//Reset complete Fifo
METHOD PROTECTED _reset : BOOL //TRUE if method is finnished
VAR_INPUT
	pMemory													: 	POINTER TO BYTE := 0;
	SizeOfMemory											: 	UDINT := 0;
END_VAR
IF pMemory = 0
	OR SizeOfMemory = 0
THEN
	_reset													:= FALSE;
	RETURN;
ELSIF TestAndSet(Interlock)
THEN
	(* delete *)
	MEMSET(pMemory,0,SizeOfMemory);
	Empty 													:= TRUE;
	Full 													:= FALSE;
	Count 													:= 0;
	_reset													:= TRUE;
	Interlock												:= FALSE;
ELSE
	_reset													:= TRUE;
END_IF
END_METHOD

END_FUNCTION_BLOCK

// POUs/DataBuffer/Fifo/FifoExt
//FifoBase extended with dynamical memory allocation
 {attribute 'enable_dynamic_creation'}
FUNCTION_BLOCK FifoExt EXTENDS FifoBase
VAR_OUTPUT CONSTANT
END_VAR   
VAR_INPUT
	MaxNoOfEntrys											: 	UDINT := 10;	//0 = dynamically allocation / <> 0 = pre allcoation of memory based on size of first entry (n * data size) 
END_VAR
VAR_OUTPUT
	pMemory													: 	POINTER TO BYTE := 0; //Pointer to memory	
	SizeOfMemory											: 	UDINT := 0; //According MaxNoOfEntrys and SizeOfData of first entry
END_VAR
VAR
	MemSizeAllocatedMemory									:	UDINT := 0; //Allocated memory 
	MemSizeOfData											:	UDINT;
	MemMaxNoOfEntrys										:	UDINT;
	ExtInterlock											:	BOOL;
END_VAR

;

METHOD PROTECTED FINAL allocate : BOOL
VAR_IN_OUT
	SizeOfData												:	UDINT;
END_VAR
VAR
	pDummy													:	POINTER TO BYTE;	
End_Var
IF pMemory = 0
THEN
	IF SizeOfData = 0 OR MaxNoOfEntrys = 0
	THEN
		Allocate											:= FALSE;	
	ELSE
		MemSizeOfData										:= SizeOfData;
		MemMaxNoOfEntrys									:= MaxNoOfEntrys;
		SizeOfMemory										:= MemSizeOfData * MemMaxNoOfEntrys;
		MemSizeAllocatedMemory								:= SizeOfMemory;
		pMemory												:= __NEW(BYTE,SizeOfMemory );
		
		IF PARAM.ENABLE_DEBUG_MSG_DYNAMIC_MEM_ALLOCATION
		THEN
			AdsLogHint('EngineeringToolbox | FB FifoExt | An instance allocated %s bytes from the dynamic memory of the ADS router memory pool', TO_STRING(SizeOfMemory));
		END_IF
	END_IF

ELSIF SizeOfData = MemSizeOfData AND MaxNoOfEntrys = MemMaxNoOfEntrys
THEN
	Allocate												:= TRUE;
	
ELSIF SizeOfData > MemSizeOfData OR MaxNoOfEntrys > MemMaxNoOfEntrys
THEN //Since increased, allocate new memory
	MemSizeAllocatedMemory									:= SizeOfData * MaxNoOfEntrys;
	pDummy													:= __NEW(BYTE, MemSizeAllocatedMemory); 
	
	 //Size of data still the same, copy old data to reuse
	IF MemSizeOfData = SizeOfData AND Count > 0
	THEN
		MEMCPY(pDummy,pMemory, SizeOfMemory);
	END_IF
	
	//Copy new settings to local variales
	MemSizeOfData											:= SizeOfData;
	MemMaxNoOfEntrys										:= MaxNoOfEntrys;	
	SizeOfMemory 											:= MemSizeAllocatedMemory;

	__DELETE(pMemory);  //Delete reference to old memory
	pMemory													:= pDummy; //Take over new pointer to new memory
	
	IF PARAM.ENABLE_DEBUG_MSG_DYNAMIC_MEM_ALLOCATION
	THEN
		AdsLogWarn('EngineeringToolbox | FB FifoExt | Value of "MaxNoOfEntrys" or data size increased and one instance allocated additional %s bytes from the dynamic memory of the ADS router memory pool', TO_STRING(SizeOfMemory));
	END_IF
	
	Allocate												:= TRUE;
	
ELSE //Size decreased
	IF MemSizeOfData <> SizeOfData AND Count > 0
	THEN //Size of data changed, erease memory 
		MEMSET(pMemory,0, MemSizeAllocatedMemory);
	ELSE //Size of data the same, keep current data
		;
	END_IF
	
	//Copy new settings to local variales
	MemSizeOfData											:= SizeOfData;
	MemMaxNoOfEntrys										:= MaxNoOfEntrys;
	SizeOfMemory											:= MemSizeOfData * MemMaxNoOfEntrys;
	Allocate												:= TRUE;
END_IF
END_METHOD

//Clear out one entry from the Fifo buffer
METHOD PUBLIC clear : BOOL //TRUE if method was successful
VAR_INPUT
	EntryNo													:	UDINT;
END_VAR             										
VAR                 										
END_VAR
Clear := SUPER^._Clear(EntryNo,This^.pMemory,This^.SizeOfMemory);
END_METHOD

//Clear out defined data set from the Fifo buffer
METHOD PUBLIC clearByDataSet : BOOL //TRUE if method was successful
VAR_INPUT
	pData													: 	POINTER TO BYTE := 0;				
END_VAR             										
VAR                 										
END_VAR
ClearByDataSet := SUPER^._ClearByDataSet(pData,SizeOfEntry,This^.pMemory,This^.SizeOfMemory);
END_METHOD

METHOD PUBLIC dequeue : BOOL //TRUE if method was successful
VAR_INPUT
	pData													:	POINTER TO BYTE;	
END_VAR
VAR
END_VAR
Dequeue := SUPER^._Dequeue(pData,SizeOfEntry,This^.pMemory,This^.SizeOfMemory);
END_METHOD

METHOD PUBLIC enqueue : BOOL //TRUE if method was successful
VAR_INPUT
	pData													:	POINTER TO BYTE;
	SizeOfData												:	UDINT;
END_VAR
VAR
	CopySize												:	UDINT;
	pDummy													:	POINTER TO BYTE;
END_VAR
IF TestAndSet(ExtInterlock) 
THEN	
	if Allocate(SizeOfData)
	then
		Enqueue 											:= SUPER^._Enqueue(pData,SizeOfData,THIS^.pMemory,THIS^.SizeOfMemory);
		ExtInterlock										:= FALSE;
	else
		Enqueue												:= FALSE;
	END_IF	
ELSE
	Enqueue													:= FALSE;
END_IF
END_METHOD

METHOD FB_exit : BOOL
VAR_INPUT
	bInCopyCode : BOOL; // if TRUE, the exit method is called for exiting an instance that is copied afterwards (online change).
END_VAR
IF NOT bInCopyCode AND pMemory <> 0
THEN //Release memory in case the PLC stopps
	__DELETE(pMemory);
	Full													:= FALSE;
	Empty													:= TRUE;
	Count													:= 0;
	SizeOfMemory											:= 0;
	MemSizeOfData											:= 0;
	MemSizeAllocatedMemory									:= 0;
	MemMaxNoOfEntrys										:= MaxNoOfEntrys;
END_IF
END_METHOD

//Check wheter a value already exist
METHOD PUBLIC isEnqueued : UDINT //pData entry exist in Fifo at idx as return value 
VAR_INPUT
	pData													: 	POINTER TO BYTE := 0;
END_VAR
IsEnqueued := SUPER^._IsEnqueued(pData,SizeOfEntry,This^.pMemory,This^.SizeOfMemory);
END_METHOD

//Check wheter a value will be the next output of the buffer
METHOD PUBLIC isNextEntry : BOOL //Inputs value is the next output 
VAR_INPUT
	pData													: 	POINTER TO BYTE := 0;
END_VAR
VAR
END_VAR
IsNextEntry := SUPER^._IsNextEntry(pData,SizeOfEntry,This^.pMemory,This^.SizeOfMemory);
END_METHOD

METHOD PUBLIC readEntry : BOOL //TRUE if method was successful
VAR_INPUT
	idx														:	UDINT;
	pData													: 	POINTER TO BYTE := 0;
END_VAR
ReadEntry := SUPER^._ReadEntry(idx,pData,SizeOfEntry,This^.pMemory,This^.SizeOfMemory);
END_METHOD

//Reset complete Fifo
METHOD PUBLIC reset : BOOL //TRUE if method is finnished
VAR_INPUT
END_VAR
reset				:= SUPER^._reset(This^.pMemory,This^.SizeOfMemory);
END_METHOD

END_FUNCTION_BLOCK

// POUs/DataBuffer/Fifo/FifoLRealSimple
//Fifo with a internal Lreal array for a simple num list implementation
FUNCTION_BLOCK FifoLRealSimple EXTENDS FifoBase
VAR_OUTPUT CONSTANT
	MIN_BUFFER												:	DINT := 1; //Fifo buffer start index 
	MAX_BUFFER												:	DINT := PARAM.FIFO_LREAL_SIMPEL_MAX_BUFFER; //Fifo buffer end index - see library parameter to customize parameter
END_VAR   
VAR_INPUT
END_VAR
VAR_OUTPUT
	Buffer													:	ARRAY[MIN_BUFFER..MAX_BUFFER] OF LREAL; //Lreal Fifo buffer 
END_VAR
VAR
END_VAR

;

 //Clear out one entry from the Fifo buffer
METHOD PUBLIC clear : BOOL //TRUE if method was successful
VAR_INPUT
	EntryNo													:	UDINT;
END_VAR             										
VAR                 										
END_VAR
Clear := super^._Clear(EntryNo,ADR(Buffer),SIZEOF(Buffer));
END_METHOD

//Clear out defined data set from the Fifo buffer
METHOD PUBLIC clearByDataSet : BOOL //TRUE if method was successful
VAR_INPUT
	Value													:	LREAL;
END_VAR             										
VAR                 										
END_VAR
ClearByDataSet := super^._ClearByDataSet(ADR(Value),SIZEOF(Value),ADR(Buffer),SIZEOF(Buffer));
END_METHOD

METHOD PUBLIC dequeue : BOOL //TRUE if method was successful
VAR_IN_OUT
	Value													:	LREAL;	
END_VAR
VAR
END_VAR
Dequeue := SUPER^._Dequeue(ADR(Value),SIZEOF(Value),ADR(Buffer),SIZEOF(Buffer));
END_METHOD

METHOD PUBLIC enqueue : BOOL //TRUE if method was successful
VAR_INPUT
	Value													:	LREAL;
END_VAR
Enqueue := SUPER^._Enqueue(ADR(Value),SIZEOF(Value),ADR(Buffer),SIZEOF(Buffer));
END_METHOD

//Check wheter a value already exist
METHOD PUBLIC isEnqueued : uDINT //In Value exist in Fifo at idx as return value  
VAR_INPUT
	Value													:	LREAL;
END_VAR
IsEnqueued := SUPER^._IsEnqueued(ADR(Value),SIZEOF(Value),ADR(Buffer),SIZEOF(Buffer));
END_METHOD

//Check wheter a value will be the next output of the buffer
METHOD PUBLIC isNextEntry : BOOL //Inputs value is the next output 
VAR_INPUT
	Value													: LREAL;
END_VAR
VAR
END_VAR
IsNextEntry := SUPER^._IsNextEntry(ADR(Value),SIZEOF(Value),ADR(Buffer),SIZEOF(Buffer));
END_METHOD

METHOD PUBLIC readEntry : BOOL //TRUE if method was successful
VAR_INPUT
	idx														:	uDINT;
END_VAR
VAR_IN_OUT
	value													: LREAL;	
END_VAR
ReadEntry := SUPER^._ReadEntry(idx,ADR(Value),SIZEOF(Value),ADR(Buffer),SIZEOF(Buffer));
END_METHOD

//Reset complete Fifo
METHOD PUBLIC reset : BOOL //TRUE if method is finnished
VAR_INPUT
END_VAR
reset := SUPER^._reset(ADR(Buffer),SIZEOF(Buffer));
END_METHOD

END_FUNCTION_BLOCK

// POUs/DataBuffer/Ringbuffer/Ringbuffer
//Ringbuffer based on external memory
FUNCTION_BLOCK Ringbuffer EXTENDS RingbufferBase
VAR_INPUT	
END_VAR
VAR_OUTPUT
END_VAR    
VAR
END_VAR

METHOD PUBLIC dequeue : BOOL //TRUE if method was successful
VAR_INPUT
	pData													: 	POINTER TO BYTE ;
	SizeOfData												: 	UDINT ;
	pMemory													: 	POINTER TO BYTE ;
	SizeOfMemory											: 	UDINT ;
END_VAR
Dequeue := SUPER^._Dequeue(pData,SizeOfData,pMemory,SizeOfMemory);
END_METHOD

METHOD PUBLIC dequeueStream : BOOL //TRUE if method was successful
VAR_INPUT
	pData													: 	POINTER TO BYTE ;
	SizeOfStream											:	UDINT ; //n * Size of last entry and not greater than SizeOfMemory
	pMemory													: 	POINTER TO BYTE;
	SizeOfMemory											: 	UDINT ;
END_VAR
VAR
END_VAR
DequeueStream := SUPER^._DequeueStream(pData,SizeOfStream,pMemory,SizeOfMemory);
END_METHOD

METHOD PUBLIC enqueue : BOOL //TRUE if method was successful
VAR_INPUT
	pData													: 	POINTER TO BYTE ;
	SizeOfData												: 	UDINT ;
	pMemory													: 	POINTER TO BYTE ;
	SizeOfMemory											: 	UDINT ;
END_VAR
Enqueue := SUPER^._Enqueue(pData,SizeOfData,pMemory,SizeOfMemory);
END_METHOD

METHOD PUBLIC enqueueStream : BOOL
VAR_INPUT
	pData													: 	POINTER TO BYTE ;
	SizeOfData												: 	UDINT ; //Size of one entry
	SizeOfStream											:	UDINT ; //n * SizeofData and not greater than SizeOfMemory
	pMemory													: 	POINTER TO BYTE ;
	SizeOfMemory											: 	UDINT ;
END_VAR
VAR
END_VAR
EnqueueStream := SUPER^._EnqueueStream(pData,SizeOfData,SizeOfStream,pMemory,SizeOfMemory);
END_METHOD

//Reset complete ring buffer
METHOD PUBLIC reset : BOOL //TRUE if method is finnished
VAR_INPUT
	pMemory													: 	POINTER TO BYTE := 0;
	SizeOfMemory											: 	UDINT := 0;
END_VAR
reset := SUPER^._reset(pMemory,SizeOfMemory);
END_METHOD

END_FUNCTION_BLOCK

// POUs/DataBuffer/Ringbuffer/RingbufferBase
//Ringbuffer basic template based on external memory
FUNCTION_BLOCK RingbufferBase
VAR_INPUT	
	Overwrite												:	BOOL := FALSE; // TRUE = overwrite oldest entry 
END_VAR
VAR_OUTPUT
	Count													:	UDINT := 0; 	// Number of entrys	
	Full													:	BOOL ;		// TRUE when max number of entrys reached
	Empty													:	BOOL := TRUE; // TRUE when no entrys present
	ReadIdx													: 	UDINT := 0;	// Read data from adress 
	WriteIdx												: 	UDINT := 0;	// Write data to adress
END_VAR    
VAR
	Interlock												:	BOOL; 
	MaxEntrys												:	UDINT; //Maximum number of entrys based on size of data and size of memory
	SizeOfEntry												:	UDINT;
	NoOfStreamEntrys										:	UDINT;
	cbData													:	UDINT;
END_VAR

METHOD PROTECTED _dequeue : BOOL //TRUE if method was successful
VAR_INPUT
	pData													: 	POINTER TO BYTE ;
	SizeOfData												: 	UDINT ;
	pMemory													: 	POINTER TO BYTE ;
	SizeOfMemory											: 	UDINT ;
END_VAR
IF 	pData = 0
	OR SizeOfData = 0
	OR pMemory = 0
	OR SizeOfMemory = 0
	OR Empty
THEN
	_Dequeue												:= FALSE;
	RETURN;
ELSIF TestAndSet(Interlock)
THEN	
	IF Count > 0
	THEN 
		(* copy dataset *)
		ReadIdx												:= ReadIdx + 1;
		IF (ReadIdx) > MaxEntrys
		THEN
			ReadIdx											:= 1;						
		END_IF
		
		MEMCPY(pData,pMemory + MAX(0, ReadIdx - 1) * SizeOfData,SizeOfData);
		
		Count 												:= MAX(0,Count - 1);
		Empty 												:= Count = 0;
		Full												:= FALSE;
		_Dequeue											:= TRUE;	
	ELSE 
		_Dequeue											:= FALSE;
	END_IF
	
	Interlock												:= FALSE;
ELSE
	_Dequeue												:= FALSE;
END_IF
END_METHOD

METHOD PROTECTED _dequeueStream : BOOL //TRUE if method was successful
VAR_INPUT
	pData													: 	POINTER TO BYTE ;
	SizeOfStream											:	UDINT ; //n * Size of last entry and not greater than SizeOfMemory
	pMemory													: 	POINTER TO BYTE;
	SizeOfMemory											: 	UDINT ;
END_VAR
VAR
END_VAR
IF 	pData = 0
	OR SizeOfEntry = 0
	OR pMemory = 0
	OR SizeOfMemory = 0
	OR Empty 
	OR SizeOfStream > SizeOfMemory
THEN
	_DequeueStream											:= FALSE;
	RETURN;
ELSIF TestAndSet(Interlock)
THEN	
	NoOfStreamEntrys										:= (SizeOfStream / SizeOfEntry); 
	IF Count > 0  
	THEN 
		(* maximum count *)
		IF ReadIdx + MIN(Count,NoOfStreamEntrys) <= MaxEntrys
		THEN //Read all data at one time
			ReadIdx											:= ReadIdx + 1; //Point to start read data			
			MEMCPY(pData,pMemory + (ReadIdx - 1) * SizeOfEntry, MIN(TO_UDINT(Count) * SizeOfEntry, SizeOfStream));
			ReadIdx											:= (ReadIdx - 1) + TO_UDINT(MIN(Count, NoOfStreamEntrys)); //Point to next index after reading x entrys
				
		ELSE //Read data with overflow					
			cbData											:= TO_UDINT(MaxEntrys) - ReadIdx; 		 
			ReadIdx											:= ReadIdx + 1; //Point to start read data	
			//Copy first part of stream our from buffer
			MEMCPY(pData, pMemory + ((ReadIdx - 1) * SizeOfEntry), cbData * SizeOfEntry );
	
			//Copy second part of stream from beginning of buffer
			ReadIdx											:= TO_UDINT(MIN(Count,NoOfStreamEntrys)) - cbData; //Point to next index after reading x entrys	
			MEMCPY( pData + (cbData * SizeOfEntry) , pMemory ,(TO_UDINT(MIN(Count,NoOfStreamEntrys)) - cbData) * SizeOfEntry);			
		END_IF
		Count 												:= MAX(0,Count - NoOfStreamEntrys);		
		Empty 												:= Count = 0;
		Full												:= FALSE;
		_DequeueStream										:= TRUE;	
		
	ELSE 
		_DequeueStream										:= FALSE;
	END_IF
	
	Interlock												:= FALSE;
ELSE
	_DequeueStream											:= FALSE;
END_IF
END_METHOD

METHOD PROTECTED _enqueue : BOOL //TRUE if method was successful
VAR_INPUT
	pData													: 	POINTER TO BYTE ;
	SizeOfData												: 	UDINT ;
	pMemory													: 	POINTER TO BYTE ;
	SizeOfMemory											: 	UDINT ;
END_VAR
IF pData = 0
	OR SizeOfData = 0
	OR pMemory = 0
	OR SizeOfMemory = 0
THEN
	_Enqueue												:= FALSE;
	RETURN;
ELSIF TestAndSet(Interlock)
THEN			
	_Enqueue												:= FALSE;
	
	(* maximum count *)
	MaxEntrys 												:= (SizeOfMemory / SizeOfData);

	IF Count < MaxEntrys OR Overwrite
	THEN
		SizeOfEntry											:= SizeOfData;
		IF MaxEntrys = Count 
		THEN //Adapt read index if write index is in front of read index
			ReadIdx											:= ReadIdx + 1;
			IF ReadIdx > TO_UDINT(MaxEntrys)
			THEN
				ReadIdx										:= 1;								
			END_IF
		END_IF	
		WriteIdx											:= WriteIdx + 1;	
		IF WriteIdx > TO_UDINT(MaxEntrys)
		THEN
			WriteIdx										:= 1;
		END_IF
	
		MEMCPY(pMemory + ((MAX(0,WriteIdx) - 1) * SizeOfData) ,pData,SizeOfData);		
		Count												:= MIN(Count + 1,  MaxEntrys);
		Full												:= Count >= MaxEntrys;
		Empty 												:= FALSE;	
		_Enqueue											:= TRUE;
	END_IF
	
	Interlock												:= FALSE;
ELSE
	_Enqueue												:= FALSE;
END_IF
END_METHOD

METHOD PROTECTED _enqueueStream : BOOL
VAR_INPUT
	pData													: 	POINTER TO BYTE ;
	SizeOfData												: 	UDINT ; //Size of one entry
	SizeOfStream											:	UDINT ; //n * SizeofData and not greater than SizeOfMemory
	pMemory													: 	POINTER TO BYTE ;
	SizeOfMemory											: 	UDINT ;
END_VAR
VAR
END_VAR
IF pData = 0
	OR SizeOfData = 0
	OR pMemory = 0
	OR SizeOfMemory = 0
	OR SizeOfStream = 0
	OR SizeOfStream > SizeOfMemory 
THEN
	_EnqueueStream											:= FALSE;
	RETURN;
ELSIF TestAndSet(Interlock)
THEN			
	_EnqueueStream											:= FALSE;
	
	(* maximum count *)
	MaxEntrys 												:= (SizeOfMemory / SizeOfData);
	SizeOfEntry												:= SizeOfData;
	NoOfStreamEntrys										:= (SizeOfStream / SizeOfData);
	
	IF (WriteIdx) + NoOfStreamEntrys <= MaxEntrys
	THEN //write full stream
		IF Count < MaxEntrys OR Overwrite
		THEN
			IF MaxEntrys = Count
			THEN //Adapt read index if write index is in front of read index
				ReadIdx										:= ReadIdx + TO_UDINT(NoOfStreamEntrys); 			
			END_IF		
		
			MEMCPY(pMemory + (WriteIdx * SizeOfData) ,pData,SizeOfStream);		
			WriteIdx										:= writeIdx + TO_UDINT(NoOfStreamEntrys);
			Count											:= MIN(Count + NoOfStreamEntrys, MaxEntrys);
			Empty 											:= FALSE;	
			_EnqueueStream									:= TRUE;
		ELSE
			_EnqueueStream									:= FALSE;
		END_IF	
	ELSIF Count + NoOfStreamEntrys <= (MaxEntrys) OR Overwrite
	THEN //Stream causes overflow
		cbData												:= TO_UDINT(MaxEntrys) - WriteIdx; 		 
		//Copy first part of stream to fill up buffer
		MEMCPY(pMemory + (WriteIdx * SizeOfData) ,pData, (cbData * SizeOfData) );	
		//Copy second part of stream to beginning of buffer
		MEMCPY(pMemory , pData + (cbData * SizeOfData) ,(TO_UDINT(NoOfStreamEntrys) - cbData) * SizeOfData);	
		
		WriteIdx											:= (writeIdx + TO_UDINT(NoOfStreamEntrys)) - TO_UDINT(MaxEntrys);
		Count												:= MIN(Count + NoOfStreamEntrys, MaxEntrys);
		IF MaxEntrys = Count
		THEN //Adapt read index if write index is in front of read index
			ReadIdx											:= WriteIdx;
		END_IF	
			
		Empty 												:= FALSE;	
		_EnqueueStream										:= TRUE;	
	ELSE
		_EnqueueStream										:= FALSE;	
	END_IF		
	Full													:= Count >= MaxEntrys;
	Interlock												:= FALSE;
ELSE
	_EnqueueStream											:= FALSE;
END_IF
END_METHOD

//Reset complete ring buffer
METHOD PROTECTED _reset : BOOL //TRUE if method is finnished
VAR_INPUT
	pMemory													: 	POINTER TO BYTE := 0;
	SizeOfMemory											: 	UDINT := 0;
END_VAR
IF pMemory = 0
	OR SizeOfMemory = 0
THEN
	_reset													:= TRUE;
	RETURN;
ELSIF TestAndSet(Interlock)
THEN
	(* delete *)
	_reset													:= TRUE;
	MEMSET(pMemory,0,SizeOfMemory);
	ReadIdx := WriteIdx										:= 0;
	Empty 													:= TRUE;
	Full													:= FALSE;
	Count 													:= 0;
	Interlock												:= FALSE;
ELSE
	_reset													:= TRUE;
END_IF
END_METHOD

END_FUNCTION_BLOCK

// POUs/DataBuffer/Ringbuffer/RingbufferByteSimple
//Ringbuffer with a internal Byte array for a simple data buffer implementation 
FUNCTION_BLOCK RingbufferByteSimple EXTENDS RingbufferBase
VAR_OUTPUT CONSTANT
	MIN_BUFFER												:	UDINT := 1; //Ringbuffer start index 
	MAX_BUFFER												:	uDINT := PARAM.RINGBUFFER_BYTE_SIMPLE_MAX_BUFFER; //Ringbuffer buffer end index - see library parameter to customize parameter
END_VAR   
VAR_INPUT
END_VAR
VAR_OUTPUT
	Buffer													:	ARRAY[MIN_BUFFER..MAX_BUFFER] OF BYTE; //Byte buffer 
END_VAR
VAR 
END_VAR

;

METHOD PUBLIC dequeue : BOOL //TRUE if method was successful
VAR_IN_OUT
	value													: BYTE;	
END_VAR
IF TestAndSet(Interlock)
THEN	
	IF Count > 0
	THEN 
		(* copy dataset *)		
		ReadIdx												:= ReadIdx + 1;
		IF (ReadIdx) > MAX_BUFFER
		THEN
			ReadIdx											:= TO_UDINT(MIN_BUFFER);				
		END_IF
		
		Value												:= Buffer[ReadIdx];
		
		Count 												:= MAX(0,Count - 1);
		Empty 												:= Count = 0;
		Full												:= FALSE;
		Dequeue												:= TRUE;	
	ELSE 
		Dequeue												:= FALSE;
	END_IF
	
	Interlock												:= FALSE;
ELSE
	Dequeue													:= FALSE;
END_IF
END_METHOD

METHOD PUBLIC dequeueStream : BOOL //TRUE if method was successful
VAR_INPUT
	pData													:	POINTER TO BYTE;
	SizeOfStream											:	UDINT;	
END_VAR
DequeueStream := super^._DequeueStream(pData, SizeOfStream,  ADR(Buffer),SIZEOF(Buffer));
END_METHOD

METHOD PUBLIC enqueue : BOOL //TRUE if method was successful
VAR_INPUT
	Value													:	BYTE;
END_VAR
IF TestAndSet(Interlock)
THEN			
	Enqueue													:= FALSE;

	IF Count < MAX_BUFFER OR Overwrite
	THEN
		IF MAX_BUFFER = Count 
		THEN //Adapt read index if write index is in front of read index
			ReadIdx											:= ReadIdx + 1;
			IF ReadIdx > TO_UDINT(MAX_BUFFER)
			THEN
				ReadIdx										:= TO_UDINT(MIN_BUFFER);							
			END_IF
		END_IF		
		WriteIdx											:= WriteIdx + 1;	
		IF WriteIdx > TO_UDINT(MAX_BUFFER)
		THEN
			WriteIdx										:= TO_UDINT(MIN_BUFFER);
		END_IF
	
		Buffer[WriteIdx]									:= Value;
	
		Count												:= MIN(Count + 1,  MAX_BUFFER);
		Full												:= Count >= MAX_BUFFER;
		Empty 												:= FALSE;	
		Enqueue												:= TRUE;
	END_IF
	
	Interlock												:= FALSE;
ELSE
	Enqueue													:= FALSE;
END_IF
END_METHOD

METHOD PUBLIC enqueueStream : BOOL //TRUE if method was successful
VAR_INPUT
	pData													:	POINTER TO BYTE;
	SizeOfStream											:	UDINT;
END_VAR
EnqueueStream := SUPER^._EnqueueStream(pData, SIZEOF(BUFFER[MIN_BUFFER] ), SizeOfStream,ADR(Buffer),SIZEOF(Buffer));
END_METHOD

//Reset complete ring buffer
METHOD PUBLIC reset : BOOL //TRUE if method is finnished
VAR_INPUT
END_VAR
reset := SUPER^._reset(ADR(Buffer),SIZEOF(Buffer));
END_METHOD

END_FUNCTION_BLOCK

// POUs/DataBuffer/Ringbuffer/RingbufferCharSimple
//Ringbuffer with a internal char array (String) for a simple num list implementation
FUNCTION_BLOCK RingbufferCharSimple EXTENDS RingbufferBase
VAR_OUTPUT CONSTANT
	MIN_BUFFER												:	UDINT := 0; //Default min index of string 
	MAX_BUFFER												:	UDINT := PARAM.RINGBUFFER_CHAR_SIMPLE_MAX_BUFFER; //Ringbuffer buffer end index - see library parameter to customize parameter
END_VAR   
VAR_INPUT
END_VAR
VAR_OUTPUT
	Buffer													:	STRING[MAX_BUFFER]; //Char buffer 
END_VAR
VAR
END_VAR

;

METHOD PUBLIC dequeue : BOOL //TRUE if method was successful
VAR_IN_OUT
	value													: BYTE;	
END_VAR
Dequeue := SUPER^._Dequeue(ADR(Value),SizeOfEntry,ADR(Buffer),SIZEOF(Buffer));
END_METHOD

METHOD PUBLIC dequeueStream : BOOL //TRUE if method was successful
VAR_INPUT
	pData													:	POINTER TO BYTE;
	SizeOfStream											:	UDINT ; //Not greater than SizeOfMemory
END_VAR
DequeueStream := SUPER^._DequeueStream(pData, SizeOfStream,  ADR(Buffer),TO_UDINT(MAX_BUFFER));
END_METHOD

METHOD PUBLIC enqueue : BOOL //TRUE if method was successful
VAR_INPUT
	Value													:	BYTE;
END_VAR
Enqueue := SUPER^._Enqueue(ADR(Value),SIZEOF(Value),ADR(Buffer),SIZEOF(Buffer));
END_METHOD

METHOD PUBLIC enqueueStream : BOOL //TRUE if method was successful
VAR_INPUT
	pData													:	POINTER TO BYTE;
	SizeOfStream											:	UDINT ; //Not greater than SizeOfMemory
END_VAR
EnqueueStream := SUPER^._EnqueueStream(pData,SIZEOF(BUFFER[MIN_BUFFER]), SizeOfStream,ADR(Buffer),TO_UDINT(MAX_BUFFER));
END_METHOD

//Reset complete ring buffer
METHOD PUBLIC reset : BOOL //TRUE if method is finnished
VAR_INPUT
END_VAR
reset := SUPER^._reset(ADR(Buffer),SIZEOF(Buffer));
END_METHOD

END_FUNCTION_BLOCK

// POUs/DataBuffer/Ringbuffer/RingbufferExt
//Ringbuffer extended with dynamical allocation of memory 
{attribute 'enable_dynamic_creation'}
FUNCTION_BLOCK RingbufferExt EXTENDS RingbufferBase
VAR_OUTPUT CONSTANT
END_VAR   
VAR_INPUT
	MaxNoOfEntrys											: 	UDINT := 10;	//0 = dynamically allocation / <> 0 = pre allcoation of memory based on size of first entry (n * data size) 
END_VAR
VAR_OUTPUT
	pMemory													: 	POINTER TO BYTE := 0;	//start address of buffer data
	SizeOfMemory											: 	UDINT := 0;	//size of buffer
END_VAR
VAR
	MemSizeAllocatedMemory									:	UDINT := 0; //Allocated memory 
	MemSizeOfData											:	UDINT;
	MemMaxNoOfEntrys										:	UDINT;
	ExtInterlock											:	BOOL;
END_VAR

;

METHOD PROTECTED FINAL allocate : BOOL
VAR_IN_OUT
	SizeOfData												:	UDINT;
END_VAR
VAR
	pDummy													:	POINTER TO BYTE;	
End_Var
IF pMemory = 0
THEN
	IF SizeOfData = 0 OR MaxNoOfEntrys = 0
	THEN
		Allocate											:= FALSE;	
	ELSE
		MemSizeOfData										:= SizeOfData;
		MemMaxNoOfEntrys									:= MaxNoOfEntrys;
		SizeOfMemory										:= MemSizeOfData * MemMaxNoOfEntrys;
		MemSizeAllocatedMemory								:= SizeOfMemory;
		pMemory												:= __NEW(BYTE,SizeOfMemory );
		
		IF PARAM.ENABLE_DEBUG_MSG_DYNAMIC_MEM_ALLOCATION
		THEN
			AdsLogHint('EngineeringToolbox | FB FifoExt | An instance allocated %s bytes from the dynamic memory of the ADS router memory pool', TO_STRING(SizeOfMemory));
		END_IF
	END_IF

ELSIF SizeOfData = MemSizeOfData AND MaxNoOfEntrys = MemMaxNoOfEntrys
THEN
	Allocate												:= TRUE;
	
ELSIF SizeOfData > MemSizeOfData OR MaxNoOfEntrys > MemMaxNoOfEntrys
THEN //Since increased, allocate new memory
	MemSizeAllocatedMemory									:= SizeOfData * MaxNoOfEntrys;
	pDummy													:= __NEW(BYTE, MemSizeAllocatedMemory); 
	
	 //Size of data still the same, copy old data to reuse
	IF MemSizeOfData = SizeOfData AND Count > 0
	THEN
		MEMCPY(pDummy,pMemory, SizeOfMemory);
	END_IF
	
	//Copy new settings to local variales
	MemSizeOfData											:= SizeOfData;
	MemMaxNoOfEntrys										:= MaxNoOfEntrys;	
	SizeOfMemory 											:= MemSizeAllocatedMemory;

	__DELETE(pMemory);  //Delete reference to old memory
	pMemory													:= pDummy; //Take over new pointer to new memory
	
	IF PARAM.ENABLE_DEBUG_MSG_DYNAMIC_MEM_ALLOCATION
	THEN
		AdsLogWarn('EngineeringToolbox | FB FifoExt | Value of "MaxNoOfEntrys" or data size increased and one instance allocated additional %s bytes from the dynamic memory of the ADS router memory pool', TO_STRING(SizeOfMemory));
	END_IF
	
	Allocate												:= TRUE;
	
ELSE //Size decreased
	IF MemSizeOfData <> SizeOfData AND Count > 0
	THEN //Size of data changed, erease memory 
		MEMSET(pMemory,0, MemSizeAllocatedMemory);
	ELSE //Size of data the same, keep current data
		;
	END_IF
	
	//Copy new settings to local variales
	MemSizeOfData											:= SizeOfData;
	MemMaxNoOfEntrys										:= MaxNoOfEntrys;
	SizeOfMemory											:= MemSizeOfData * MemMaxNoOfEntrys;
	Allocate												:= TRUE;
END_IF
END_METHOD

METHOD PUBLIC dequeue : BOOL //TRUE if method was successful
VAR_INPUT
	pData													:	POINTER TO BYTE;	
END_VAR
VAR
END_VAR
Dequeue := SUPER^._Dequeue(pData,SizeOfEntry,This^.pMemory,This^.SizeOfMemory);
END_METHOD

METHOD PUBLIC dequeueStream : BOOL //TRUE if method was successful
VAR_INPUT
	pData													:	POINTER TO BYTE;	
	SizeOfStream											:	UDINT ; //Not greater than SizeOfMemory
END_VAR
VAR
END_VAR
DequeueStream := SUPER^._DequeueStream(pData,SizeOfStream , This^.pMemory,This^.SizeOfMemory);
END_METHOD

METHOD PUBLIC enqueue : BOOL //TRUE if method was successful
VAR_INPUT
	pData													:	POINTER TO BYTE;
	SizeOfData												:	UDINT;
END_VAR
VAR
END_VAR
IF TestAndSet(ExtInterlock) 
THEN	
	if Allocate(SizeOfData)
	then
		Enqueue 											:= SUPER^._Enqueue(pData,SizeOfData,THIS^.pMemory,THIS^.SizeOfMemory);
		ExtInterlock										:= FALSE;
	else
		Enqueue												:= FALSE;
	END_IF	
ELSE
	Enqueue													:= FALSE;
END_IF
END_METHOD

METHOD PUBLIC enqueueStream : BOOL //TRUE if method was successful
VAR_INPUT
	pData													:	POINTER TO BYTE;
	SizeOfData												:	UDINT; //Size of one entry
	SizeOfStream											:	UDINT ; //Not greater than SizeOfMemory
END_VAR
VAR
END_VAR
IF TestAndSet(ExtInterlock) 
THEN	
	if Allocate(SizeOfData)
	then
		EnqueueStream 										:= SUPER^._EnqueueStream(pData,SizeOfData,SizeOfStream,THIS^.pMemory,THIS^.SizeOfMemory);
		ExtInterlock										:= FALSE;
	else
		EnqueueStream										:= FALSE;
	END_IF	
ELSE
	EnqueueStream											:= FALSE;
END_IF
END_METHOD

METHOD FB_exit : BOOL
VAR_INPUT
	bInCopyCode : BOOL; // if TRUE, the exit method is called for exiting an instance that is copied afterwards (online change).
END_VAR
IF NOT bInCopyCode AND pMemory <> 0
THEN //Release memory in case the PLC stopps
	__DELETE(pMemory);
	SizeOfMemory								:= 0;
END_IF
END_METHOD

//Reset complete ring buffer
METHOD PUBLIC reset : BOOL //TRUE if method is finnished
VAR_INPUT
END_VAR
IF pMemory = 0
THEN //no memroy allocated
	reset													:= TRUE;
ELSE //Just delte the memory
	reset 													:= SUPER^._reset(THIS^.pMemory,THIS^.SizeOfMemory);	
END_IF
END_METHOD

END_FUNCTION_BLOCK

// POUs/DataBuffer/Ringbuffer/RingbufferLRealSimple
//Ringbuffer with a internal Lreal array for a simple num list implementation 
FUNCTION_BLOCK RingbufferLRealSimple EXTENDS RingbufferBase
VAR_OUTPUT CONSTANT
	MIN_BUFFER												:	UDINT := 1; //Ringbuffer start index
	MAX_BUFFER												:	UDINT := PARAM.RINGBUFFER_LREAL_SIMPLE_MAX_BUFFER; //Ringbuffer buffer end index - see library parameter to customize parameter
END_VAR   
VAR_INPUT
END_VAR
VAR_OUTPUT
	Buffer													:	ARRAY[MIN_BUFFER..MAX_BUFFER] OF LREAL; //Lreal buffer 
END_VAR
VAR 
END_VAR

;

METHOD PUBLIC dequeue : BOOL //TRUE if method was successful
VAR_IN_OUT
	value													: LREAL;	
END_VAR
Dequeue := SUPER^._Dequeue(ADR(Value),SizeOfEntry,ADR(Buffer),SIZEOF(Buffer));
END_METHOD

METHOD PUBLIC dequeueStream : BOOL //TRUE if method was successful
VAR_INPUT
	pData													:	POINTER TO LREAL;
	SizeOfStream											:	UDINT ; //Not greater than SizeOfMemory
END_VAR
DequeueStream := super^._DequeueStream(pData,SizeOfStream,  ADR(Buffer),SIZEOF(Buffer));
END_METHOD

METHOD PUBLIC enqueue : BOOL //TRUE if method was successful
VAR_INPUT
	Value													:	LREAL;
END_VAR
Enqueue := SUPER^._Enqueue(ADR(Value),SIZEOF(Value),ADR(Buffer),SIZEOF(Buffer));
END_METHOD

METHOD PUBLIC enqueueStream : BOOL //TRUE if method was successful
VAR_INPUT
	pData													:	POINTER TO LREAL;
	SizeOfStream											:	UDINT ; //Not greater than SizeOfMemory
END_VAR
EnqueueStream := SUPER^._EnqueueStream(pData,SIZEOF(BUFFER[MIN_BUFFER]), SizeOfStream,ADR(Buffer),SIZEOF(Buffer));
END_METHOD

//Reset complete ring buffer
METHOD PUBLIC reset : BOOL //TRUE if method is finnished
VAR_INPUT
END_VAR
reset := SUPER^._reset(ADR(Buffer),SIZEOF(Buffer));
END_METHOD

END_FUNCTION_BLOCK

// POUs/DataBuffer/DataFileLogger
{attribute 'no_check' := ''}
//Extension to FB "DoubleBuffer" to write the recorded data cyclic into a file 
{attribute 'enable_dynamic_creation'}
FUNCTION_BLOCK DataFileLogger EXTENDS DoubleBuffer
VAR_OUTPUT CONSTANT 
	{attribute 'displaymode':='binary'}
	OPTION_KEEP_FILE_ON_ERROR								: 	BYTE := 2#0000_0001; //Keep file open in error case to be able to contine after reset
	{attribute 'displaymode':='binary'}
	OPTION_START_WITH_NEW_FILE								: 	BYTE := 2#1000_0000; //Create empty file with enable flag instead open and continue existing file
END_VAR                     								
VAR_INPUT                   								
	Enable													: 	BOOL; //Enable to write looked data cyclic into file  
	ResetTrig												: 	BOOL; //Reset internal error 

{attribute 'displaymode':='binary'}
	Options													: 	BYTE := 2#00000000; // See outputs constant OPTION_xxx
	Path													: 	STRING := 'C:\temp'; //Path and filename
	Filetype												: 	STRING(6) := '.log'; //file tpye
END_VAR                     								
VAR_IN_OUT                  								
END_VAR                     								
VAR_OUTPUT       
	TimeWriteFile											:	TIME; //Elapsed time to write data to file 
	hFile													: 	UINT; //Current file handle
	Busy													: 	BOOL; //Write msg to file active   
	Error													: 	BOOL;     
	{attribute 'displaymode':='hex'}   								
	ErrorId													: 	UDINT; //Ads error Id of file handling function blocks or HRESULT (hr) ADS error code 
END_VAR                     								
VAR            
//local ************************************************************************************
	WriteCounter											:	UDINT; //Endless write counter fyi
	State													: 	INT;
	StartTimeWriteData										:	TIME;			

//trigger *********************************************************************************

//timer ***********************************************************************************

//instances ***********************************************************************************             								
	FILEOPEN												: 	FB_FileOpen := (sNetId:='',tTimeout:=DEFAULT_ADS_TIMEOUT, ePath:=PATH_GENERIC);
	FILECLOSE												: 	FB_FileClose := (sNetId:='',tTimeout:=DEFAULT_ADS_TIMEOUT);
	FILEWRITE												: 	FB_FileWrite := (sNetId:='',tTimeout:=DEFAULT_ADS_TIMEOUT);

//Dummys ****************************************************************************************

END_VAR

	(* Data file logger based on two buffer concept 		*)
	(********************************************************)

(* Sequence started by method addData if buffer is filled ***************************************************)
	CASE State OF
	0:	
		IF Error
		THEN
			IF ResetTrig OR NOT Enable
			THEN
				Error										:= FALSE;
				ErrorId										:= 0;
				hr											:= S_OK;

				FileOpen(bExecute:=FALSE);	
				FileClose(bExecute:=FALSE);	
				FILEWRITE(bExecute:=FALSE);
			ELSIF NOT OPtions.0 AND hFile <> 0	
			THEN
				FileClose(bExecute:=TRUE , hFile := hFile);
				State										:= 3;
			END_IF
			
		ELSIF Enable
		THEN
			IF hr <> S_OK
			THEN //Method executed with error
				Error										:= TRUE;
				ErrorId										:= HRESULT_TO_ADSERROR(hr);
			ELSIF hFile = 0
			THEN
				WriteCounter								:= 0;	
				FileOpen(bExecute:= TRUE , sPathName:= CONCAT(Path,Filetype), nMode:=SEL(Options.7 ,FOPEN_MODEAPPEND,FOPEN_MODEWRITE) OR FOPEN_MODETEXT OR FOPEN_MODEPLUS );
				State										:= 1;		
			ELSIF ReadyToRead
			THEN
				FILEWRITE(bExecute:=TRUE ,hFile:= hFile , pWriteBuff := pDataToRead, cbWriteLen := SizeOfDataToRead);
				StartTimeWriteData							:= TIME();
				State										:= 2;			
			END_IF
		
		ELSIF hFile <> 0
		THEN //Not enabled
			IF NOT Empty
			THEN //Write rest of buffer		
				IF NOT ReadyToRead THEN setReadyToRead(TRUE); END_IF 
				FILEWRITE(bExecute:=ReadyToRead ,hFile:= hFile , pWriteBuff := pDataToRead, cbWriteLen := SizeOfDataToRead);
				StartTimeWriteData							:= TIME();
				State										:= 2;
			ELSE
				FileClose(bExecute:=TRUE , hFile := hFile);
				state										:= 3;	
			END_IF
        END_IF
     
	(* Open file *******************************************************************************)                                          	
	1:                       	
		FileOpen();                                     	
		IF NOT FileOpen.bBusy                           	
		THEN                                            	
			IF FileOpen.bError                          	
			THEN            
				Error										:= TRUE;                            	
				ErrorId										:= FileOpen.nErrId;
				State										:= 0;
			ELSE                                     	
				hFile										:= FileOpen.hFile;
				IF ReadyToRead
				THEN //Write request acitive
					FILEWRITE(bExecute:=TRUE ,hFile:= hFile , pWriteBuff := pDataToRead, cbWriteLen := SizeOfDataToRead);
					StartTimeWriteData						:= TIME();
					State									:= 2;
				ELSE
					State									:= 0;
				END_IF			
			END_IF
			FileOpen(bExecute:=FALSE);			
		END_IF

	(* Write data to file **********************************************************************)
	2: 
		FILEWRITE(hFile:= hFile);	
		IF NOT FILEWRITE.bBusy
		THEN
			IF FILEWRITE.bError
			THEN
				Error										:= TRUE;       
				ErrorId										:= FILEWRITE.nErrId;
				state										:= 0;
			ELSE                            
				WriteCounter								:= WriteCounter + 1;
				TimeWriteFile								:= TIME() - StartTimeWriteData;          	
				State										:= 0;	
			END_IF	
			setReadyToRead(FALSE); 
			FILEWRITE(bExecute:=FALSE);          		
		END_IF

	(* Close File ******************************************************************************)
	3: 
		FileClose(hFile := hFile);
		IF NOT FileClose.bBusy
		THEN
			IF FileClose.bError
			THEN
				Error										:= TRUE;       
				ErrorId										:= FileClose.nErrId;
				State										:= 0;
			ELSE                                        		
				hFile										:= 0;
				State										:= 0;
			END_IF
			FileClose(bExecute:=FALSE);
		END_IF
	ELSE
		;
	END_CASE

(* Ack ErrorIds **********************************************************)
	Busy 													:= State <> 0;
(**************************************************************************)

METHOD PUBLIC addData : HRESULT //Add data into write buffer and swap if if buffer is filled
VAR_INPUT
	pData													:	POINTER TO BYTE;
	SizeofData												:	UDINT;
END_VAR
IF NOT Error
THEN 
	IF SUPER^.addData(pData,SizeOfData) <> S_OK
	THEN
		ErrorId												:= HRESULT_TO_ADSERROR(hr);
		Error												:= TRUE;
	END_IF
ELSE
	addData													:= SEL(Error , E_HRESULTADSERR.INVALIDACCESS ,E_HRESULTADSERR.ERROR);
END_IF
END_METHOD

METHOD PUBLIC addString : HRESULT //Add string to write buffer and swap if buffer is filled
VAR_INPUT
	Data													:	T_MAXSTRING;
END_VAR
addString := This^.addData(ADR(Data),TO_UDINT(LEN(Data)));
END_METHOD

PROPERTY PUBLIC optKeepFileOnError : BOOL
GET
optKeepFileOnError := Options.0;
END_GET
SET
Options.0				:= optKeepFileOnError;
END_SET
END_PROPERTY

PROPERTY PUBLIC optStartNewFile : BOOL
GET
optStartNewFile := Options.7;
END_GET
SET
Options.7				:= optStartNewFile;
END_SET
END_PROPERTY

END_FUNCTION_BLOCK

// POUs/DataBuffer/DoubleBuffer
//Double buffer FB to fill one part of buffer while the other (filled) part can be read or processed meanwhile
//Variable "ReadyToRead" signals that recorded data can be read consistent by pointer "pDataToRead" 
//After the data are processed or copied, it is needed to call the method "setReadyToReady(Status := FALSE)" and release the buffer to be used if the other half is filled 
//With setReadyToReady(Status := TRUE) you can mark the current write buffer as "ReadyToRead" on demand and accessible via "pDataToRead"  (e.g. if no more data need to be recorded)
{attribute 'enable_dynamic_creation'}
FUNCTION_BLOCK DoubleBuffer
VAR_OUTPUT CONSTANT 	
END_VAR                     								
VAR_INPUT
	Overwrite												:	BOOL ; //Overwrite buffer read buffer if not released -> setReadyToRead(FALSE)        
	SizeOfMemory											: 	UDINT := 5120;	//Total size of dynamic allocated buffer (will be splited in half)	   								
END_VAR                     								
VAR_IN_OUT                  								
END_VAR                     								
VAR_OUTPUT       
	TimeFillBuffer											: 	TIME; //Last elapsed time to fill the buffer and set ReadyToRead=TRUE
	Full													:	BOOL; //Buffer is full
	Empty													:	BOOL := TRUE; //Buffer is empty 
	ReadyToRead												:	BOOL; //TRUE = Data are ready and can be read via "pDataToRead" to process 
	pDataToRead												:	POINTER TO BYTE; //Pointer to recorded data/filled buffer	
	SizeOfDataToRead										:	UDINT; //Count of bytes in filled buffer ready to ready 
{attribute 'displaymode':='hex'}
	hr														:	HRESULT; //Last result of method call
END_VAR                     								
VAR            
//local ************************************************************************************
	Interlock												:	BOOL; //Task interlock
	Buffer2Active											:	BOOL; //Indicates active buffer pointer 
	pBuffer1												: 	POINTER TO BYTE; //Pointer to start of allocated memory
	pBuffer2												: 	POINTER TO BYTE; //Pointer to second half of allocated memory
	StartTimeFillBuffer										:	TIME;

	MemSizeOfAllocatedMemory								: 	UDINT; //Total size of allocated memory
	MemSizeOfBuffer											: 	UDINT; //Size of split buffer
	MemSizeOfWriteBuffer									:	UDINT; //Actual size of recorded data


//trigger *********************************************************************************

//timer ***********************************************************************************

//instances ***********************************************************************************             								

//Dummys ****************************************************************************************

END_VAR

METHOD PUBLIC addData : HRESULT //Add data to write buffer and sets "ReadyToRead" if buffer is filled and data can be read to process 
VAR_INPUT
	pData													:	POINTER TO BYTE;
	SizeofData												:	UDINT;
END_VAR

IF pData <> 0 
THEN		
	//Allocate Memory to buffer messages
	IF pBuffer1 = 0
		OR SizeOfMemory > MemSizeOfAllocatedMemory 
	THEN //Allocate full memory with first entry 		
		IF NOT Allocate(SizeOfMemory)
		THEN
			addData := hr										:= E_HRESULTADSERR.NOMEMORY;
			RETURN;														
		END_IF					
	END_IF	

	IF MemSizeOfWriteBuffer = 0 THEN StartTimeFillBuffer := TIME(); END_IF
	
	//Change buffer if filled
	IF SizeofData + MemSizeOfWriteBuffer >= MemSizeOfBuffer
	THEN
		IF setReadyToRead(TRUE) <> S_OK
		THEN
			addData 											:= hr;
			RETURN;
		END_IF
	ELSE
		Full													:= FALSE;
		Empty													:= FALSE;
	END_IF
			
	//Copy data to buffer
	MEMCPY(SEL(Buffer2Active, pBuffer1, pBuffer2) + MemSizeOfWriteBuffer, pData, SizeofData);
	MemSizeOfWriteBuffer										:= MemSizeOfWriteBuffer + SizeofData;
	
	addData := hr												:= S_OK;
ELSE
	addData := hr												:= E_HRESULTADSERR.INVALIDPARM;
END_IF
END_METHOD

METHOD PUBLIC addString : HRESULT //Add string to write buffer and sets "ReadyToRead" if buffer is filled and data can be read to process 
VAR_INPUT
	Data													:	T_MAXSTRING;
END_VAR
addString := hr := addData(ADR(Data),TO_UDINT(LEN(Data)));
END_METHOD

METHOD PROTECTED FINAL allocate : BOOL //allocte buffer memory form router pool
VAR_INPUT
	SizeOfBuffer											:	UDINT;
END_VAR
VAR
	pDummy													:	POINTER TO BYTE;	
End_Var
IF SizeOfBuffer	= 0
THEN
	Allocate												:= FALSE;
	
ELSIF pBuffer1 = 0
THEN
	MemSizeOfAllocatedMemory								:= SizeOfBuffer;
	pBuffer1												:= __NEW(BYTE,MemSizeOfAllocatedMemory );
	MemSizeOfBuffer											:= MemSizeOfAllocatedMemory / 2;
	pBuffer2												:= pBuffer1 + MemSizeOfBuffer; 
	Buffer2Active											:= FALSE;
	MemSizeOfWriteBuffer									:= 0;
	
	IF PARAM.ENABLE_DEBUG_MSG_DYNAMIC_MEM_ALLOCATION
	THEN
		AdsLogHint('EngineeringToolbox | FB DoubleBuffer | An instance allocated %s bytes from the dynamic memory of the ADS router memory pool', TO_STRING(MemSizeOfAllocatedMemory));
	END_IF	
	Allocate												:= TRUE;
ELSIF SizeOfBuffer > MemSizeOfBuffer 
THEN //Since increased, allocate new memory
	
	pDummy													:= __NEW(BYTE, SizeOfBuffer); 

	IF SizeOfBuffer > MemSizeOfAllocatedMemory
	THEN //Size increased rescue data from old memory
		IF Buffer2Active
		THEN
			MEMCPY(pDummy,pBuffer2, MemSizeOfBuffer);
		ELSE
			MEMCPY(pDummy,pBuffer1, MemSizeOfBuffer);	
		END_IF
	END_IF

	__DELETE(pBuffer1);  //Delete reference to old memory
	
	MemSizeOfAllocatedMemory								:= SizeOfBuffer;
	pBuffer1												:= pDummy; //Take over new pointer to new memory
	Buffer2Active											:= FALSE;
	MemSizeOfBuffer											:= MemSizeOfAllocatedMemory / 2;
	pBuffer2												:= pBuffer1 + MemSizeOfBuffer; 
	MemSizeOfWriteBuffer										:= 0;
	
	IF PARAM.ENABLE_DEBUG_MSG_DYNAMIC_MEM_ALLOCATION
	THEN
		AdsLogWarn('EngineeringToolbox | FB DoubleBuffer | Value of "SizeOfMemory" increased and an instance has an additional %s bytes allocated from the dynamic memory of the ADS router memory pool', TO_STRING(MemSizeOfAllocatedMemory));
	END_IF
	
	Allocate												:= TRUE;
	
ELSE //Size decreased
	Allocate												:= TRUE;
END_IF
END_METHOD

METHOD PUBLIC copyData : HRESULT //Copy data from buffer (pDataToRead) into destination and reset "ReadyToReady" back to false if succeful executed 
VAR_INPUT
	pDest													:	POINTER TO BYTE; 
	SizeOfDest												:	UDINT; //Size of destination/data to copy
END_VAR
IF pDest <> 0 AND SizeOfDest > 0
	AND pDataToRead <> 0 
THEN
	MEMCPY(pDest, pDataToRead, MIN(SizeOfDest,SizeOfDataToRead));										
	hr		 												:= setReadyToRead(FALSE);	
	
ELSE
	IF pDataToRead = 0
	THEN
		hr													:= E_HRESULTADSERR.NOTREADY;
	ELSIF pDest = 0 
	THEN 
		hr													:= E_HRESULTADSERR.INVALIDPARM;
	ELSIF SizeOfDest = 0
	THEN
		hr													:= E_HRESULTADSERR.INVALIDPARM;	
	END_IF
END_IF
copyData													:= hr;
END_METHOD

METHOD FB_exit : BOOL
VAR_INPUT
	bInCopyCode : BOOL; // if TRUE, the exit method is called for exiting an instance that is copied afterwards (online change).
END_VAR
IF NOT bInCopyCode AND pBuffer1 <> 0
THEN //Release memory in case the PLC stopps
	__DELETE(pBuffer1);
END_IF
END_METHOD

{attribute 'monitoring' := 'call'}
PROPERTY PUBLIC fillLevel : INT //Buffer fill level 100% if both parts of buffer are filled
GET
IF MemSizeOfBuffer <> 0
THEN
	fillLevel												:= 	TO_INT((50.0 / TO_LREAL(MemSizeOfBuffer)) * TO_LREAL(MemSizeOfWriteBuffer))
																+ SEL(ReadyToRead, 0, TO_INT((50.0 / TO_LREAL(MemSizeOfBuffer)) * TO_LREAL(SizeOfDataToRead)));
ELSE
	fillLevel												:= 0;
END_IF
END_GET
END_PROPERTY

//Reset buffer 
METHOD PUBLIC reset : BOOL //TRUE if method is finnished
VAR_INPUT
END_VAR
TimeFillBuffer												:= T#0MS;
Full														:= FALSE; //Buffer is full
Empty														:= TRUE; //Buffer is empty 
ReadyToRead													:= FALSE;
SizeOfDataToRead											:= 0;
hr															:= S_OK;
MemSizeOfWriteBuffer										:= 0;
reset														:= TRUE;
END_METHOD

METHOD PUBLIC setReadyToRead : HRESULT //Status = FALSE to reset "ReadyToRead" and unlock buffer / Status = TRUE to mark current write buffer as filled and "ReadyToRead", accessible via "pDataToRead"
VAR_INPUT
	Status								:	BOOL; //FALSE to reset "ReadyToRead" or TRUE to set "ReadyToRead" and swap buffer 
END_VAR
IF TestAndSet(Interlock)
THEN
	IF NOT Status
	THEN
		ReadyToRead									:= FALSE;
		Full										:= FALSE;
		Empty										:= MemSizeOfWriteBuffer = 0;
		hr											:= S_OK;
	ELSIF Overwrite 
		OR NOT ReadyToRead
	THEN //Set ready to ready and swap buffer
		hr											:= SEL(swapBuffer(), E_HRESULTADSERR.ABORTED ,S_OK);
		ReadyToRead									:= SizeOfDataToRead > 0;
		Full										:= FALSE;
		Empty										:= NOT ReadyToRead;
	ELSE
		Full										:= TRUE;
		Empty										:= FALSE;
		hr											:= E_HRESULTADSERR.ABORTED;	
	END_IF
		
	setReadyToRead									:= hr;
	Interlock										:= FALSE;
ELSE
	setReadyToRead									:= E_HRESULTADSERR.BUSY;
END_IF
END_METHOD

METHOD PROTECTED FINAL swapBuffer : BOOL //swap write and read buffer and asign filled buffer to pDataToRead
VAR_INPUT
END_VAR
pDataToRead													:= SEL(Buffer2Active, pBuffer1, pBuffer2);
SizeOfDataToRead											:= MemSizeOfWriteBuffer;	

Buffer2Active												:= NOT Buffer2Active;	

MemSizeOfWriteBuffer										:= 0;
TimeFillBuffer												:= TIME() - StartTimeFillBuffer;
StartTimeFillBuffer											:= TIME();
swapBuffer													:= TRUE;
END_METHOD

END_FUNCTION_BLOCK

// POUs/DataBuffer/Quicksort
// this funktionblock sorts an array of struct by an contained element with quicksort routine
// Udpate: compare with static PivotElement
// Find Explanation under https://www.youtube.com/watch?v=eNUM23f6g-s&ab_channel=Studyflix
{attribute 'enable_dynamic_creation'}
FUNCTION_BLOCK Quicksort
VAR CONSTANT
	MAX_STRING_LENGTH										:	INT := PARAM.QUICKSORT_MAX_STRING_LENGTH;
	MAX_WSTRING_LENGTH										:	INT := PARAM.QUICKSORT_MAX_WSTRING_LENGTH;
END_VAR
VAR_INPUT
	SortInverse												:	BOOL := FALSE;//inverses order of content
	IgnoreBlank												:	BOOL := FALSE;//sort blank characters at last			
END_VAR
VAR_OUTPUT
END_VAR
VAR
	pElement_Tmp											:	POINTER TO BYTE;		// Copy Pointer 3 - allocated memory
	MemSizeOfStruct											:	UDINT;
END_VAR

;

METHOD PROTECTED FINAL allocate : BOOL
VAR_INPUT
	SizeOfStruct											: 	UDINT;	
END_VAR
IF SizeOfStruct = 0
THEN
	allocate												:= FALSE;
ELSIF pElement_Tmp = 0 
THEN
	pElement_Tmp											:= __NEW(BYTE, SizeOfStruct);
	MemSizeOfStruct											:= SizeOfStruct;
	IF TRUE
	THEN
		AdsLogHint('EngineeringToolbox | FB Quicksort | An instance allocated %s bytes from the dynamic memory of the ADS router memory pool', TO_STRING(MemSizeOfStruct));
	END_IF
	Allocate												:= TRUE;
ELSIF SizeOfStruct > MemSizeOfStruct
THEN
	__DELETE(pElement_Tmp);	
	pElement_Tmp											:= __NEW(BYTE, SizeOfStruct);
	MemSizeOfStruct											:= SizeOfStruct;
		IF TRUE
	THEN
		AdsLogWarn('EngineeringToolbox | FB Quicksort | SizeOfStruct increased and an instance has an additional %s bytes allocated from the dynamic memory of the ADS router memory pool', TO_STRING(MemSizeOfStruct));
	END_IF
	Allocate												:= TRUE;
ELSE
	Allocate												:= TRUE;	
END_IF
END_METHOD

METHOD byDINT : BOOL // returns true if sort ends successfully 
VAR_INPUT
	pData													: 	POINTER TO BYTE := 0;	// ADR(Array) 	
	SizeOfData												: 	UDINT := 0;				// SIZEOF(Array)
	pCompareElement											: 	POINTER TO BYTE := 0;	// ADR(Array[1].DINT)		
	SizeOfStruct											: 	UDINT := 0;				// SIZEOF(Array[1]) 	
END_VAR                                                 
VAR        
	pPivotElement											: 	POINTER TO DINT;		// Pivot value
	PivotElement											: 	DINT;					// Pivot value as DINT	
	pCmpElement												:	POINTER TO DINT;		// compare value
	                                					                            	
	endMainLoop												:	BOOL;					// End of main loop reached
	endSubLoop												:	BOOL;					// End of sub loop reached                                              
	ElementCount											:	DINT;					// No of array elements
	stackCount,left,right,i,j								:	DINT;					// running variables 	
	stack													:	ARRAY[1..32] OF UDINT;	// stack size 32 => ~1 Mio elements *)	
	                                					
	pElement_1												:	POINTER TO BYTE;		// Copy Pointer 1		
	pElement_2												:	POINTER TO BYTE;		// Copy Pointer 2

END_VAR
// ends with true in case of no error	                                    					 					
IF SizeOfStruct = 0 OR SizeOfData = 0
	OR pData = 0 OR pCompareElement = 0
THEN               					                                   					
	byDINT													:= FALSE;
	RETURN;   
ELSE
	byDINT													:= TRUE;                          					
END_IF                                  					
          
// calculate no. of Elements                                
ElementCount												:= TO_DINT(SizeOfData / SizeOfStruct);   		
			
// Quicksort                            					
// initial value of array size          					
left 														:= 1;				// first element
right 														:= ElementCount;	// last element 
stackCount 													:= 1;				// running variable 
                                        	
WHILE NOT endMainLoop DO							
	IF left < right THEN                	
		pPivotElement										:= pCompareElement + (SizeOfStruct * TO_UDINT(SHR(right+left,1)));
		PivotElement										:= pPivotElement^;
		i 													:= left -1;
		j 													:= right +1;
		endSubLoop 											:= FALSE;
		REPEAT
			IF SortInverse
			THEN	// sort descending	
				REPEAT	
					i 										:= i+1;	
					pCmpElement								:= pCompareElement + (SizeOfStruct * TO_UDINT(i-1));
				UNTIL (pCmpElement^ <= PivotElement) OR NOT (i < right)	END_REPEAT	
				REPEAT	
					j 										:= j-1;	
					pCmpElement								:= pCompareElement + (SizeOfStruct * TO_UDINT(j-1));
				UNTIL (pCmpElement^ >= PivotElement) OR NOT (j > left)	END_REPEAT		
			ELSE	// sort ascending
				REPEAT	
					i 										:= i+1;
					pCmpElement								:= pCompareElement + (SizeOfStruct * TO_UDINT(i-1));
				UNTIL (pCmpElement^ >= PivotElement)	OR NOT (i < right)	END_REPEAT;				
				REPEAT	
					j 										:= j-1;	
					pCmpElement								:= pCompareElement + (SizeOfStruct * TO_UDINT(j-1));
				UNTIL (pCmpElement^ <= PivotElement) OR NOT (j > left)	END_REPEAT;
			END_IF
			IF i >= j THEN
				endSubLoop									:= TRUE;
			ELSE                    					
				Allocate( SizeOfStruct);
				pElement_1									:= pData + (SizeOfStruct * TO_UDINT(j-1));
				pElement_2									:= pData + (SizeOfStruct * TO_UDINT(i-1));
				
				IF pElement_Tmp = 0 
					OR_ELSE MEMCPY(pElement_Tmp, pElement_1,	SizeOfStruct) = 0
					OR_ELSE MEMCPY(pElement_1,	pElement_2,		SizeOfStruct) = 0
					OR_ELSE MEMCPY(pElement_2,	pElement_Tmp,	SizeOfStruct) = 0
				THEN
					byDINT									:= FALSE;
					RETURN;	
				END_IF
	
			END_IF
		UNTIL endSubLoop END_REPEAT;		
		stack[stackCount] 									:= TO_UDINT(right); 	// save right in stack			
		IF stackCount < 32              					
		THEN                            					
			stackCount 										:= stackCount +1;
		ELSE															// Error stack Limit    
			endMainLoop 									:= TRUE;
			byDINT											:= FALSE;			
		END_IF                          					
		right 												:= MAX(left, i-1);
	ELSE                                
		IF stackCount = 1 THEN          
			endMainLoop 									:= TRUE;
		ELSE                            					
			left 											:= right+1;       
			stackCount 										:= stackCount -1;	// load from stack
			right											:= TO_DINT(stack[stackCount]);
		END_IF
	END_IF
END_WHILE
END_METHOD

METHOD byDINT_Bubble : BOOL // returns true if sort ends successfully 
VAR_INPUT	
	pData													:	POINTER TO BYTE;// ADR(Array) 			
	SizeOfData												:	UDINT;			// SIZEOF(Array)
	pCompareElement											:	POINTER TO BYTE;// ADR(Array[1].DINT)		
	SizeOfStruct											:	UDINT;			// SIZEOF(Array[1]) 			
END_VAR                                 					                
VAR                                     					                
	Run  													:	DINT;			// main loop
  	Index													:	DINT;			// sub loop 	
	ElementCount											:	DINT;			
	                                    					
	CompareElement_1										:	DINT;					
	CompareElement_2										:	DINT;					
	pCompareElement_1										:	POINTER TO DINT;		
	pCompareElement_2										:	POINTER TO DINT;
		                                					                        
	pElement_1												:	POINTER TO BYTE;		
	pElement_2												:	POINTER TO BYTE;		
END_VAR
// ends with true in case of no error	                                    					 					
IF SizeOfStruct = 0 OR SizeOfData = 0
	OR pData = 0 OR pCompareElement = 0
THEN               					                                   					
	byDINT_Bubble											:= FALSE;
	RETURN;   
ELSE
	byDINT_Bubble											:= TRUE;                          					
END_IF    

// Bubblesort Routine
// Code saving 
	
// calculate no. of Elements                                
ElementCount												:= TO_DINT(SizeOfData / SizeOfStruct);  

// bubblesort 
FOR Run := 1 TO TO_DINT(ElementCount) - 1 DO
    FOR Index := ElementCount - 1 TO Run BY -1 DO
		// get element x for compare 
		pCompareElement_1				:=	pCompareElement + (SizeOfStruct * TO_UDINT(Index));
		CompareElement_1				:=	pCompareElement_1^;
		// get element x-1 for compare 
		pCompareElement_2				:=	pCompareElement + (SizeOfStruct * TO_UDINT(Index-1));
		CompareElement_2 				:=	pCompareElement_2^;
		// switch by useing temporary memory 
		IF ((	CompareElement_1 < CompareElement_2) AND NOT SortInverse)
			OR((CompareElement_1 > CompareElement_2) AND SortInverse)
		THEN
			// get pointer for MEMCPY 
			Allocate(SizeOfStruct);
			pElement_1					:= pData + SizeOfStruct * TO_UDINT(Index);
			pElement_2					:= pData + SizeOfStruct * TO_UDINT(Index-1);
			
	
			IF pElement_Tmp = 0 
				OR_ELSE MEMCPY(pElement_Tmp, pElement_1,	SizeOfStruct) = 0
				OR_ELSE MEMCPY(pElement_1,	pElement_2,		SizeOfStruct) = 0
				OR_ELSE MEMCPY(pElement_2,	pElement_Tmp,	SizeOfStruct) = 0
			THEN
				byDINT_Bubble		:= FALSE;
				EXIT;												
			END_IF

      END_IF
	END_FOR
END_FOR
END_METHOD

METHOD byINT : BOOL // returns true if sort ends successfully 
VAR_INPUT
	pData													: 	POINTER TO BYTE := 0;	// ADR(Array) 	
	SizeOfData												: 	UDINT := 0;				// SIZEOF(Array)
	pCompareElement											: 	POINTER TO BYTE := 0;	// ADR(Array[1].INT)		
	SizeOfStruct											: 	UDINT := 0;				// SIZEOF(Array[1]) 	
END_VAR                                                 
VAR        
	pPivotElement											: 	POINTER TO INT;			// Pivot value
	PivotElement											: 	INT;					// Pivot value as INT	
	pCmpElement												:	POINTER TO INT;			// compare value
	                                					                            	
	endMainLoop												:	BOOL;					// End of main loop reached
	endSubLoop												:	BOOL;					// End of sub loop reached                                              
	ElementCount											:	DINT;					// No of array elements
	stackCount,left,right,i,j								:	DINT;					// running variables 	
	stack													:	ARRAY[1..32] OF UDINT;	// stack size 32 => ~1 Mio elements *)	
	                                					
	pElement_1												:	POINTER TO BYTE;		// Copy Pointer 1		
	pElement_2												:	POINTER TO BYTE;		// Copy Pointer 2
END_VAR
// ends with true in case of no error	                                    					 					
IF SizeOfStruct = 0 OR SizeOfData = 0
	OR pData = 0 OR pCompareElement = 0
THEN               					                                   					
	byINT													:= FALSE;
	RETURN;   
ELSE
	byINT													:= TRUE;                          					
END_IF                                    					
        
// calculate no. of Elements                                
ElementCount												:= TO_DINT(SizeOfData / SizeOfStruct);   
                                					
// Quicksort                            					
// initial value of array size          					
left 														:= 1;				// first element
right 														:= ElementCount;	// last element 
stackCount 													:= 1;				// running variable 
                                        	
WHILE NOT endMainLoop DO							
	IF left < right THEN                	
		pPivotElement										:= pCompareElement + (SizeOfStruct * TO_UDINT(SHR(right+left,1)));
		PivotElement										:= pPivotElement^;
		i 													:= left -1;
		j 													:= right +1;
		endSubLoop 											:= FALSE;
		REPEAT
			IF SortInverse
			THEN	// sort descending	
				REPEAT	
					i 										:= i+1;	
					pCmpElement								:= pCompareElement + (SizeOfStruct * TO_UDINT(i-1));
				UNTIL (pCmpElement^ <= PivotElement) OR NOT (i < right)	END_REPEAT	
				REPEAT	
					j 										:= j-1;	
					pCmpElement								:= pCompareElement + (SizeOfStruct * TO_UDINT(j-1));
				UNTIL (pCmpElement^ >= PivotElement) OR NOT (j > left)	END_REPEAT		
			ELSE	// sort ascending
				REPEAT	
					i 										:= i+1;
					pCmpElement								:= pCompareElement + (SizeOfStruct * TO_UDINT(i-1));
				UNTIL (pCmpElement^ >= PivotElement)	OR NOT (i < right)	END_REPEAT;				
				REPEAT	
					j 										:= j-1;	
					pCmpElement								:= pCompareElement + (SizeOfStruct * TO_UDINT(j-1));
				UNTIL (pCmpElement^ <= PivotElement) OR NOT (j > left)	END_REPEAT;
			END_IF
			IF i >= j THEN
				endSubLoop									:= TRUE;
			ELSE                    					
				Allocate(SizeOfStruct);
				pElement_1									:= pData + (SizeOfStruct * TO_UDINT(j-1));
				pElement_2									:= pData + (SizeOfStruct * TO_UDINT(i-1));
				
				IF pElement_Tmp = 0 
					OR_ELSE MEMCPY(pElement_Tmp, pElement_1,	SizeOfStruct) = 0
					OR_ELSE MEMCPY(pElement_1,	pElement_2,		SizeOfStruct) = 0
					OR_ELSE MEMCPY(pElement_2,	pElement_Tmp,	SizeOfStruct) = 0
				THEN
					byINT									:= FALSE;
					RETURN;	
				END_IF
	
			END_IF
		UNTIL endSubLoop END_REPEAT;		
		stack[stackCount] 									:= TO_UDINT(right); 	// save right in stack			
		IF stackCount < 32              					
		THEN                            					
			stackCount 										:= stackCount +1;
		ELSE															// Error stack Limit    
			endMainLoop 									:= TRUE;
			byINT											:= FALSE;			
		END_IF                          					
		right 												:= MAX(left, i-1);
	ELSE                                
		IF stackCount = 1 THEN          
			endMainLoop 									:= TRUE;
		ELSE                            					
			left 											:= right+1;       
			stackCount 										:= stackCount -1;	// load from stack
			right											:= TO_DINT(stack[stackCount]);
		END_IF
	END_IF
END_WHILE
END_METHOD

METHOD byLREAL : BOOL // returns true if sort ends successfully 
VAR_INPUT
	pData													: 	POINTER TO BYTE := 0;	// ADR(Array) 	
	SizeOfData												: 	UDINT := 0;				// SIZEOF(Array)
	pCompareElement											: 	POINTER TO BYTE := 0;	// ADR(Array[1].LREAL)		
	SizeOfStruct											: 	UDINT := 0;				// SIZEOF(Array[1]) 	
END_VAR                                                 
VAR        
	pPivotElement											: 	POINTER TO LREAL;		// Pivot value	
	PivotElement											: 	LREAL;					// Pivot value as LREAL
	pCmpElement												:	POINTER TO LREAL;		// compare value
	                                					                            	
	endMainLoop												:	BOOL;					// End of main loop reached
	endSubLoop												:	BOOL;					// End of sub loop reached                                              
	ElementCount											:	DINT;					// No of array elements
	stackCount,left,right,i,j								:	DINT;					// running variables 	
	stack													:	ARRAY[1..32] OF UDINT;	// stack size 32 => ~1 Mio elements *)	
	                                					
	pElement_1												:	POINTER TO BYTE;		// Copy Pointer 1		
	pElement_2												:	POINTER TO BYTE;		// Copy Pointer 2
	
END_VAR
// ends with true in case of no error	                                    					 					
IF SizeOfStruct = 0 OR SizeOfData = 0
	OR pData = 0 OR pCompareElement = 0
THEN               					                                   					
	byLREAL													:= FALSE;
	RETURN;   
ELSE
	byLREAL													:= TRUE;                          					
END_IF                                 					
            
// calculate no. of Elements                                
ElementCount												:= TO_DINT(SizeOfData / SizeOfStruct);   
                            					
// Quicksort                            					
// initial value of array size          					
left 														:= 1;				// first element
right 														:= ElementCount;	// last element 
stackCount 													:= 1;				// running variable 
                                        	
WHILE NOT endMainLoop DO							
	IF left < right THEN                	
		pPivotElement										:= pCompareElement + (SizeOfStruct * TO_UDINT(SHR(right+left,1))); // divide by 2
		PivotElement										:= pPivotElement^;
		i 													:= left -1;
		j 													:= right +1;
		endSubLoop 											:= FALSE;
		REPEAT
			IF SortInverse
			THEN	// sort descending	
				REPEAT	
					i 										:= i+1;	
					pCmpElement								:= pCompareElement + (SizeOfStruct * TO_UDINT(i-1));
				UNTIL (pCmpElement^ <= PivotElement) OR NOT (i < right)	END_REPEAT	
				REPEAT	
					j 										:= j-1;	
					pCmpElement								:= pCompareElement + (SizeOfStruct * TO_UDINT(j-1));
				UNTIL (pCmpElement^ >= PivotElement) OR NOT (j > left)	END_REPEAT		
			ELSE	// sort ascending
				REPEAT	
					i 										:= i+1;
					pCmpElement								:= pCompareElement + (SizeOfStruct * TO_UDINT(i-1));
				UNTIL (pCmpElement^ >= PivotElement)	OR NOT (i < right)	END_REPEAT;				
				REPEAT	
					j 										:= j-1;	
					pCmpElement								:= pCompareElement + (SizeOfStruct * TO_UDINT(j-1));
				UNTIL (pCmpElement^ <= PivotElement) OR NOT (j > left)	END_REPEAT;
			END_IF
			IF i >= j THEN
				endSubLoop									:= TRUE;
			ELSE                    					
				Allocate(SizeOfStruct);
				pElement_1									:= pData + (SizeOfStruct * TO_UDINT(j-1));
				pElement_2									:= pData + (SizeOfStruct * TO_UDINT(i-1));
				
				IF pElement_Tmp = 0 
					OR_ELSE MEMCPY(pElement_Tmp, pElement_1,	SizeOfStruct) = 0
					OR_ELSE MEMCPY(pElement_1,	pElement_2,		SizeOfStruct) = 0
					OR_ELSE MEMCPY(pElement_2,	pElement_Tmp,	SizeOfStruct) = 0
				THEN
					byLREAL									:= FALSE;
					RETURN;	
				END_IF

			END_IF
		UNTIL endSubLoop END_REPEAT;		
		stack[stackCount] 									:= TO_UDINT(right); 	// save right in stack			
		IF stackCount < 32              					
		THEN                            					
			stackCount 										:= stackCount +1;
		ELSE															// Error stack Limit    
			endMainLoop 									:= TRUE;
			byLREAL											:= FALSE;			
		END_IF                          					
		right 												:= MAX(left, i-1);
	ELSE                                
		IF stackCount = 1 THEN          
			endMainLoop 									:= TRUE;
		ELSE                            					
			left 											:= right+1;       
			stackCount 										:= stackCount -1;	// load from stack
			right											:= TO_DINT(stack[stackCount]);
		END_IF
	END_IF
END_WHILE
END_METHOD

METHOD byLTIME : BOOL // returns true if sort ends successfully 
VAR_INPUT
	pData													: 	POINTER TO BYTE := 0;	// ADR(Array) 	
	SizeOfData												: 	UDINT := 0;				// SIZEOF(Array)
	pCompareElement											: 	POINTER TO BYTE := 0;	// ADR(Array[1].LTIME)		
	SizeOfStruct											: 	UDINT := 0;				// SIZEOF(Array[1]) 	
END_VAR                                                 
VAR        
	pPivotElement											: 	POINTER TO LTIME;		// Pivot value	
	PivotElement											: 	LTIME;					// Pivot value as LTIME	
	pCmpElement												:	POINTER TO LTIME;		// compare value
	                                					                            	
	endMainLoop												:	BOOL;					// End of main loop reached
	endSubLoop												:	BOOL;					// End of sub loop reached                                              
	ElementCount											:	DINT;					// No of array elements
	stackCount,left,right,i,j								:	DINT;					// running variables 	
	stack													:	ARRAY[1..32] OF UDINT;	// stack size 32 => ~1 Mio elements *)	
	                                					
	pElement_1												:	POINTER TO BYTE;		// Copy Pointer 1		
	pElement_2												:	POINTER TO BYTE;		// Copy Pointer 2
END_VAR
// ends with true in case of no error	                                    					 					
IF SizeOfStruct = 0 OR SizeOfData = 0
	OR pData = 0 OR pCompareElement = 0
THEN               					                                   					
	byLTIME													:= FALSE;
	RETURN;   
ELSE
	byLTIME													:= TRUE;                          					
END_IF                                    					
             
// calculate no. of Elements                                
ElementCount												:= TO_DINT(SizeOfData / SizeOfStruct);   
                           					
// Quicksort                            					
// initial value of array size          					
left 														:= 1;				// first element
right 														:= ElementCount;	// last element 
stackCount 													:= 1;				// running variable 
                                        	
WHILE NOT endMainLoop DO							
	IF left < right THEN                	
		pPivotElement										:= pCompareElement + (SizeOfStruct * TO_UDINT(SHR(right+left,1)));
		PivotElement										:= pPivotElement^;
		i 													:= left -1;
		j 													:= right +1;
		endSubLoop 											:= FALSE;
		REPEAT
			IF SortInverse
			THEN	// sort descending	
				REPEAT	
					i 										:= i+1;	
					pCmpElement								:= pCompareElement + (SizeOfStruct * TO_UDINT(i-1));
				UNTIL (pCmpElement^ <= PivotElement) OR NOT (i < right)	END_REPEAT	
				REPEAT	
					j 										:= j-1;	
					pCmpElement								:= pCompareElement + (SizeOfStruct * TO_UDINT(j-1));
				UNTIL (pCmpElement^ >= PivotElement) OR NOT (j > left)	END_REPEAT		
			ELSE	// sort ascending
				REPEAT	
					i 										:= i+1;
					pCmpElement								:= pCompareElement + (SizeOfStruct * TO_UDINT(i-1));
				UNTIL (pCmpElement^ >= PivotElement)	OR NOT (i < right)	END_REPEAT;				
				REPEAT	
					j 										:= j-1;	
					pCmpElement								:= pCompareElement + (SizeOfStruct * TO_UDINT(j-1));
				UNTIL (pCmpElement^ <= PivotElement) OR NOT (j > left)	END_REPEAT;
			END_IF
			IF i >= j THEN
				endSubLoop									:= TRUE;
			ELSE                    					
				Allocate(SizeOfStruct);
				pElement_1									:= pData + (SizeOfStruct * TO_UDINT(j-1));
				pElement_2									:= pData + (SizeOfStruct * TO_UDINT(i-1));
				
				IF pElement_Tmp = 0 
					OR_ELSE MEMCPY(pElement_Tmp, pElement_1,	SizeOfStruct) = 0
					OR_ELSE MEMCPY(pElement_1,	pElement_2,		SizeOfStruct) = 0
					OR_ELSE MEMCPY(pElement_2,	pElement_Tmp,	SizeOfStruct) = 0
				THEN
					byLTIME									:= FALSE;
					RETURN;	
				END_IF

			END_IF
		UNTIL endSubLoop END_REPEAT;		
		stack[stackCount] 									:= TO_UDINT(right); 	// save right in stack			
		IF stackCount < 32              					
		THEN                            					
			stackCount 										:= stackCount +1;
		ELSE															// Error stack Limit    
			endMainLoop 									:= TRUE;
			byLTIME											:= FALSE;			
		END_IF                          					
		right 												:= MAX(left, i-1);
	ELSE                                
		IF stackCount = 1 THEN          
			endMainLoop 									:= TRUE;
		ELSE                            					
			left 											:= right+1;       
			stackCount 										:= stackCount -1;	// load from stack
			right											:= TO_DINT(stack[stackCount]);
		END_IF
	END_IF
END_WHILE
END_METHOD

METHOD byREAL : BOOL // returns true if sort ends successfully 
VAR_INPUT
	pData													: 	POINTER TO BYTE := 0;	// ADR(Array) 	
	SizeOfData												: 	UDINT := 0;				// SIZEOF(Array)
	pCompareElement											: 	POINTER TO BYTE := 0;	// ADR(Array[1].REAL)		
	SizeOfStruct											: 	UDINT := 0;				// SIZEOF(Array[1]) 	
END_VAR                                                 
VAR        
	pPivotElement											: 	POINTER TO REAL;		// Pivot value	
	PivotElement											: 	REAL;					// Pivot value as REAL	
	pCmpElement												:	POINTER TO REAL;		// compare value
	                                					                            	
	endMainLoop												:	BOOL;					// End of main loop reached
	endSubLoop												:	BOOL;					// End of sub loop reached                                              
	ElementCount											:	DINT;					// No of array elements
	stackCount,left,right,i,j								:	DINT;					// running variables 	
	stack													:	ARRAY[1..32] OF UDINT;	// stack size 32 => ~1 Mio elements *)	
	                                					
	pElement_1												:	POINTER TO BYTE;		// Copy Pointer 1		
	pElement_2												:	POINTER TO BYTE;		// Copy Pointer 2
END_VAR
// ends with true in case of no error	                                    					 					
IF SizeOfStruct = 0 OR SizeOfData = 0
	OR pData = 0 OR pCompareElement = 0
THEN               					                                   					
	byREAL													:= FALSE;
	RETURN;   
ELSE
	byREAL													:= TRUE;                          					
END_IF                                   					
          
// calculate no. of Elements                                
ElementCount												:= TO_DINT(SizeOfData / SizeOfStruct);   
                              					
// Quicksort                            					
// initial value of array size          					
left 														:= 1;				// first element
right 														:= ElementCount;	// last element 
stackCount 													:= 1;				// running variable 
                                        	
WHILE NOT endMainLoop DO							
	IF left < right THEN                	
		pPivotElement										:= pCompareElement + (SizeOfStruct * TO_UDINT(SHR(right+left,1)));
		PivotElement										:= pPivotElement^;
		i 													:= left -1;
		j 													:= right +1;
		endSubLoop 											:= FALSE;
		REPEAT
			IF SortInverse
			THEN	// sort descending	
				REPEAT	
					i 										:= i+1;	
					pCmpElement								:= pCompareElement + (SizeOfStruct * TO_UDINT(i-1));
				UNTIL (pCmpElement^ <= PivotElement) OR NOT (i < right)	END_REPEAT	
				REPEAT	
					j 										:= j-1;	
					pCmpElement								:= pCompareElement + (SizeOfStruct * TO_UDINT(j-1));
				UNTIL (pCmpElement^ >= PivotElement) OR NOT (j > left)	END_REPEAT		
			ELSE	// sort ascending
				REPEAT	
					i 										:= i+1;
					pCmpElement								:= pCompareElement + (SizeOfStruct * TO_UDINT(i-1));
				UNTIL (pCmpElement^ >= PivotElement)	OR NOT (i < right)	END_REPEAT;				
				REPEAT	
					j 										:= j-1;	
					pCmpElement								:= pCompareElement + (SizeOfStruct * TO_UDINT(j-1));
				UNTIL (pCmpElement^ <= PivotElement) OR NOT (j > left)	END_REPEAT;
			END_IF
			IF i >= j THEN
				endSubLoop									:= TRUE;
			ELSE                    					
				Allocate(SizeOfStruct);
				pElement_1									:= pData + (SizeOfStruct * TO_UDINT(j-1));
				pElement_2									:= pData + (SizeOfStruct * TO_UDINT(i-1));
				
				IF pElement_Tmp = 0 
					OR_ELSE MEMCPY(pElement_Tmp, pElement_1,	SizeOfStruct) = 0
					OR_ELSE MEMCPY(pElement_1,	pElement_2,		SizeOfStruct) = 0
					OR_ELSE MEMCPY(pElement_2,	pElement_Tmp,	SizeOfStruct) = 0
				THEN
					byREAL									:= FALSE;
					RETURN;	
				END_IF

			END_IF
		UNTIL endSubLoop END_REPEAT;		
		stack[stackCount] 									:= TO_UDINT(right); 	// save right in stack			
		IF stackCount < 32              					
		THEN                            					
			stackCount 										:= stackCount +1;
		ELSE															// Error stack Limit    
			endMainLoop 									:= TRUE;
			byREAL											:= FALSE;			
		END_IF                          					
		right 												:= MAX(left, i-1);
	ELSE                                
		IF stackCount = 1 THEN          
			endMainLoop 									:= TRUE;
		ELSE                            					
			left 											:= right+1;       
			stackCount 										:= stackCount -1;	// load from stack
			right											:= TO_DINT(stack[stackCount]);
		END_IF
	END_IF
END_WHILE
END_METHOD

METHOD bySTRING : BOOL // returns true if sort ends successfully 
VAR_INPUT
	pData													: 	POINTER TO BYTE := 0;	// ADR(Array) 	
	SizeOfData												: 	UDINT := 0;				// SIZEOF(Array)
	pCompareElement											: 	POINTER TO BYTE := 0;	// ADR(Array[1].STRING)		
	SizeOfStruct											: 	UDINT := 0;				// SIZEOF(Array[1]) 	
END_VAR                                                                                        
VAR        
	pPivotElement											: 	POINTER TO STRING(MAX_STRING_LENGTH);	// Pivot value
	pCmpElement												:	POINTER TO STRING(MAX_STRING_LENGTH);	// compare value
	PivotElement											:	BYTE; 					// Pivot value	
	CompareElement											:	BYTE; 					// compare value
                               					                            	
	endMainLoop												:	BOOL;					// End of main loop reached
	endSubLoop												:	BOOL;					// End of sub loop reached                                              
	ElementCount											:	DINT;					// No of array elements
	stackCount,left,right,i,j,k								:	DINT;					// running variables 	
	stack													:	ARRAY[1..32] OF UDINT;	// stack size 32 => ~1 Mio elements *)	
	                                					
	pElement_1												:	POINTER TO BYTE;		// Copy Pointer 1		
	pElement_2												:	POINTER TO BYTE;		// Copy Pointer 2
END_VAR
// ends with true in case of no error	                                    					 					
IF SizeOfStruct = 0 OR SizeOfData = 0
	OR pData = 0 OR pCompareElement = 0
THEN               					                                   					
	bySTRING												:= FALSE;
	RETURN;   
ELSE
	bySTRING												:= TRUE;                          					
END_IF                                 					
          
// calculate no. of Elements                                
ElementCount												:= TO_DINT(SizeOfData / SizeOfStruct);   
                              					
// Quicksort                            					
// initial value of array size          					
left 														:= 1;				// first element
right 														:= ElementCount;	// last element 
stackCount 													:= 1;				// running variable 
                                        	
WHILE NOT endMainLoop DO							
	IF left < right THEN                	
		pPivotElement										:= pCompareElement + (SizeOfStruct * TO_UDINT(SHR(right+left,1)));
		i 													:= left -1;
		j 													:= right +1;
		endSubLoop 											:= FALSE;
		REPEAT
			IF SortInverse
			THEN	// sort descending	
				REPEAT	
					i 										:= i+1;	
					pCmpElement								:= pCompareElement + (SizeOfStruct * TO_UDINT(i-1));
					FOR k := 1 TO MAX_STRING_LENGTH DO // Find unequal char
						// element 1,2 to upper char 	https://www.uni-due.de/hummell/infos/ascii/
						IF pCmpElement^[k] = 0 
							AND IgnoreBlank
						THEN
							CompareElement					:= 127;
						ELSE
							CompareElement					:= SEL(pCmpElement^[k] >= 97(*a*)	AND_THEN pCmpElement^[k] <= 122(*z*), 	pCmpElement^[k],pCmpElement^[k] - 32);		// a --> A
						END_IF						
						IF pPivotElement^[k] = 0 
							AND IgnoreBlank
						THEN
							PivotElement					:= 127;
						ELSE
							PivotElement					:= SEL(pPivotElement^[k] >= 97(*a*) AND_THEN pPivotElement^[k] <= 122(*z*), pPivotElement^[k], 	pPivotElement^[k] - 32);// a --> A
						END_IF
						// Find unequal char
						IF CompareElement <> PivotElement
							OR CompareElement = 0
							OR PivotElement = 0
						THEN
							EXIT;
						END_IF
					END_FOR
				UNTIL (CompareElement <= PivotElement) OR NOT (i < right)	END_REPEAT	
				REPEAT	
					j 										:= j-1;	
					pCmpElement								:= pCompareElement + (SizeOfStruct * TO_UDINT(j-1));
					FOR k := 0 TO MAX_STRING_LENGTH DO // Find unequal char
						// element 1,2 to upper char 	https://www.uni-due.de/hummell/infos/ascii/
						IF pCmpElement^[k] = 0 
							AND IgnoreBlank
						THEN
							CompareElement					:= 127;
						ELSE
							CompareElement					:= SEL(pCmpElement^[k] >= 97(*a*)	AND_THEN pCmpElement^[k] <= 122(*z*), 	pCmpElement^[k],pCmpElement^[k] - 32);		// a --> A
						END_IF
						IF pPivotElement^[k] = 0 
							AND IgnoreBlank
						THEN
							PivotElement					:= 127;
						ELSE
							PivotElement					:= SEL(pPivotElement^[k] >= 97(*a*) AND_THEN pPivotElement^[k] <= 122(*z*), pPivotElement^[k], 	pPivotElement^[k] - 32);// a --> A
						END_IF
						// Find unequal char
						IF CompareElement <> PivotElement
							OR CompareElement = 0
							OR PivotElement = 0
						THEN
							EXIT;
						END_IF
					END_FOR
				UNTIL (CompareElement >= PivotElement) OR NOT (j > left)	END_REPEAT		
			ELSE	// sort ascending
				REPEAT	
					i 										:= i+1;
					pCmpElement								:= pCompareElement + (SizeOfStruct * TO_UDINT(i-1));
					FOR k := 0 TO MAX_STRING_LENGTH DO // Find unequal char
						// element 1,2 to upper char 	https://www.uni-due.de/hummell/infos/ascii/
						IF pCmpElement^[k] = 0 
							AND IgnoreBlank
						THEN
							CompareElement					:= 127;
						ELSE
							CompareElement					:= SEL(pCmpElement^[k] >= 97(*a*)	AND_THEN pCmpElement^[k] <= 122(*z*), 	pCmpElement^[k],pCmpElement^[k] - 32);		// a --> A
						END_IF
						IF pPivotElement^[k] = 0 
							AND IgnoreBlank
						THEN
							PivotElement					:= 127;
						ELSE
							PivotElement					:= SEL(pPivotElement^[k] >= 97(*a*) AND_THEN pPivotElement^[k] <= 122(*z*), pPivotElement^[k], 	pPivotElement^[k] - 32);// a --> A
						END_IF
						// Find unequal char
						IF CompareElement <> PivotElement
							OR CompareElement = 0
							OR PivotElement = 0
						THEN
							EXIT;
						END_IF
					END_FOR
				UNTIL (CompareElement >= PivotElement)	OR NOT (i < right)	END_REPEAT;				
				REPEAT	
					j 										:= j-1;	
					pCmpElement								:= pCompareElement + (SizeOfStruct * TO_UDINT(j-1));
					FOR k := 0 TO MAX_STRING_LENGTH DO // Find unequal char
						// element 1,2 to upper char 	https://www.uni-due.de/hummell/infos/ascii/
						IF pCmpElement^[k] = 0 
							AND IgnoreBlank
						THEN	
							CompareElement					:= 127;
						ELSE
							CompareElement					:= SEL(pCmpElement^[k] >= 97(*a*)	AND_THEN pCmpElement^[k] <= 122(*z*), 	pCmpElement^[k],pCmpElement^[k] - 32);		// a --> A
						END_IF
						IF pPivotElement^[k] = 0
							AND IgnoreBlank 
						THEN
							PivotElement					:= 127;
						ELSE
							PivotElement					:= SEL(pPivotElement^[k] >= 97(*a*) AND_THEN pPivotElement^[k] <= 122(*z*), pPivotElement^[k], 	pPivotElement^[k] - 32);// a --> A
						END_IF
						// Find unequal char
						IF CompareElement <> PivotElement
							OR CompareElement = 0
							OR PivotElement = 0
						THEN
							EXIT;
						END_IF
					END_FOR
				UNTIL (CompareElement <= PivotElement) OR NOT (j > left)	END_REPEAT;
			END_IF
			IF i >= j THEN
				endSubLoop									:= TRUE;
			ELSE                    					
				Allocate(SizeOfStruct);
				pElement_1									:= pData + (SizeOfStruct * TO_UDINT(j-1));
				pElement_2									:= pData + (SizeOfStruct * TO_UDINT(i-1));
				
				IF pElement_Tmp = 0 
					OR_ELSE MEMCPY(pElement_Tmp, pElement_1,	SizeOfStruct) = 0
					OR_ELSE MEMCPY(pElement_1,	pElement_2,		SizeOfStruct) = 0
					OR_ELSE MEMCPY(pElement_2,	pElement_Tmp,	SizeOfStruct) = 0
				THEN
					bySTRING								:= FALSE;
					RETURN;	
				END_IF

			END_IF
		UNTIL endSubLoop END_REPEAT;		
		stack[stackCount] 									:= TO_UDINT(right); 	// save right in stack			
		IF stackCount < 32              					
		THEN                            					
			stackCount 										:= stackCount +1;
		ELSE															// Error stack Limit    
			endMainLoop 									:= TRUE;
			bySTRING										:= FALSE;			
		END_IF                          					
		right 												:= MAX(left, i-1);
	ELSE                                
		IF stackCount = 1 THEN          
			endMainLoop 									:= TRUE;
		ELSE                            					
			left 											:= right+1;       
			stackCount 										:= stackCount -1;	// load from stack
			right											:= TO_DINT(stack[stackCount]);
		END_IF
	END_IF
END_WHILE
END_METHOD

METHOD byTIME : BOOL // returns true if sort ends successfully 
VAR_INPUT
	pData													: 	POINTER TO BYTE := 0;	// ADR(Array) 	
	SizeOfData												: 	UDINT := 0;				// SIZEOF(Array)
	pCompareElement											: 	POINTER TO BYTE := 0;	// ADR(Array[1].TIME)		
	SizeOfStruct											: 	UDINT := 0;				// SIZEOF(Array[1]) 	
END_VAR                                                 
VAR        
	pPivotElement											: 	POINTER TO TIME;		// Pivot value
	PivotElement											: 	TIME;					// Pivot value as TIME	
	pCmpElement												:	POINTER TO TIME;		// compare value
	                                					                            	
	endMainLoop												:	BOOL;					// End of main loop reached
	endSubLoop												:	BOOL;					// End of sub loop reached                                              
	ElementCount											:	DINT;					// No of array elements
	stackCount,left,right,i,j								:	DINT;					// running variables 	
	stack													:	ARRAY[1..32] OF UDINT;	// stack size 32 => ~1 Mio elements *)	
	                                					
	pElement_1												:	POINTER TO BYTE;		// Copy Pointer 1		
	pElement_2												:	POINTER TO BYTE;		// Copy Pointer 2
END_VAR
// ends with true in case of no error	                                    					 					
IF SizeOfStruct = 0 OR SizeOfData = 0
	OR pData = 0 OR pCompareElement = 0
THEN               					                                   					
	byTIME													:= FALSE;
	RETURN;   
ELSE
	byTIME													:= TRUE;                          					
END_IF   

// calculate no. of Elements                                
ElementCount												:= TO_DINT(SizeOfData / SizeOfStruct);                                   					
                                        					
// Quicksort                            					
// initial value of array size          					
left 														:= 1;				// first element
right 														:= ElementCount;	// last element 
stackCount 													:= 1;				// running variable 
                                        	
WHILE NOT endMainLoop DO							
	IF left < right THEN                	
		pPivotElement										:= pCompareElement + (SizeOfStruct * TO_UDINT(SHR(right+left,1)));
		PivotElement										:= pPivotElement^;
		i 													:= left -1;
		j 													:= right +1;
		endSubLoop 											:= FALSE;
		REPEAT
			IF SortInverse
			THEN	// sort descending	
				REPEAT	
					i 										:= i+1;	
					pCmpElement								:= pCompareElement + (SizeOfStruct * TO_UDINT(i-1));
				UNTIL (pCmpElement^ <= PivotElement) OR NOT (i < right)	END_REPEAT	
				REPEAT	
					j 										:= j-1;	
					pCmpElement								:= pCompareElement + (SizeOfStruct * TO_UDINT(j-1));
				UNTIL (pCmpElement^ >= PivotElement) OR NOT (j > left)	END_REPEAT		
			ELSE	// sort ascending
				REPEAT	
					i 										:= i+1;
					pCmpElement								:= pCompareElement + (SizeOfStruct * TO_UDINT(i-1));
				UNTIL (pCmpElement^ >= PivotElement)	OR NOT (i < right)	END_REPEAT;				
				REPEAT	
					j 										:= j-1;	
					pCmpElement								:= pCompareElement + (SizeOfStruct * TO_UDINT(j-1));
				UNTIL (pCmpElement^ <= PivotElement) OR NOT (j > left)	END_REPEAT;
			END_IF
			IF i >= j THEN
				endSubLoop									:= TRUE;
			ELSE                    					
				Allocate(SizeOfStruct);
				pElement_1									:= pData + (SizeOfStruct * TO_UDINT(j-1));
				pElement_2									:= pData + (SizeOfStruct * TO_UDINT(i-1));
				
				IF pElement_Tmp = 0 
					OR_ELSE MEMCPY(pElement_Tmp, pElement_1,	SizeOfStruct) = 0
					OR_ELSE MEMCPY(pElement_1,	pElement_2,		SizeOfStruct) = 0
					OR_ELSE MEMCPY(pElement_2,	pElement_Tmp,	SizeOfStruct) = 0
				THEN
					byTIME									:= FALSE;
					RETURN;	
				END_IF

			END_IF
		UNTIL endSubLoop END_REPEAT;		
		stack[stackCount] 									:= TO_UDINT(right); 	// save right in stack			
		IF stackCount < 32              					
		THEN                            					
			stackCount 										:= stackCount +1;
		ELSE															// Error stack Limit    
			endMainLoop 									:= TRUE;
			byTIME											:= FALSE;			
		END_IF                          					
		right 												:= MAX(left, i-1);
	ELSE                                
		IF stackCount = 1 THEN          
			endMainLoop 									:= TRUE;
		ELSE                            					
			left 											:= right+1;       
			stackCount 										:= stackCount -1;	// load from stack
			right											:= TO_DINT(stack[stackCount]);
		END_IF
	END_IF
END_WHILE
END_METHOD

METHOD byUINT : BOOL // returns true if sort ends successfully 
VAR_INPUT
	pData													: 	POINTER TO BYTE := 0;	// ADR(Array) 	
	SizeOfData												: 	UDINT := 0;				// SIZEOF(Array)
	pCompareElement											: 	POINTER TO BYTE := 0;	// ADR(Array[1].UINT)		
	SizeOfStruct											: 	UDINT := 0;				// SIZEOF(Array[1]) 	
END_VAR                                                 
VAR        
	pPivotElement											: 	POINTER TO UINT;		// Pivot value	
	PivotElement											: 	UINT;					// Pivot value as UINT	
	pCmpElement												:	POINTER TO UINT;		// compare value
	                                					                            	
	endMainLoop												:	BOOL;					// End of main loop reached
	endSubLoop												:	BOOL;					// End of sub loop reached                                              
	ElementCount											:	DINT;					// No of array elements
	stackCount,left,right,i,j								:	DINT;					// running variables 	
	stack													:	ARRAY[1..32] OF UDINT;	// stack size 32 => ~1 Mio elements *)	
	                                					
	pElement_1												:	POINTER TO BYTE;		// Copy Pointer 1		
	pElement_2												:	POINTER TO BYTE;		// Copy Pointer 2
END_VAR
// ends with true in case of no error	                                    					 					
IF SizeOfStruct = 0 OR SizeOfData = 0
	OR pData = 0 OR pCompareElement = 0
THEN               					                                   					
	byUINT													:= FALSE;
	RETURN;   
ELSE
	byUINT													:= TRUE;                          					
END_IF     

// calculate no. of Elements                                
ElementCount												:= TO_DINT(SizeOfData / SizeOfStruct);                                 					
                                        					
// Quicksort                            					
// initial value of array size          					
left 														:= 1;				// first element
right 														:= ElementCount;	// last element 
stackCount 													:= 1;				// running variable 
                                        	
WHILE NOT endMainLoop DO							
	IF left < right THEN                	
		pPivotElement										:= pCompareElement + (SizeOfStruct * TO_UDINT(SHR(right+left,1)));
		PivotElement										:= pPivotElement^;
		i 													:= left -1;
		j 													:= right +1;
		endSubLoop 											:= FALSE;
		REPEAT
			IF SortInverse
			THEN	// sort descending	
				REPEAT	
					i 										:= i+1;	
					pCmpElement								:= pCompareElement + (SizeOfStruct * TO_UDINT(i-1));
				UNTIL (pCmpElement^ <= PivotElement) OR NOT (i < right)	END_REPEAT	
				REPEAT	
					j 										:= j-1;	
					pCmpElement								:= pCompareElement + (SizeOfStruct * TO_UDINT(j-1));
				UNTIL (pCmpElement^ >= PivotElement) OR NOT (j > left)	END_REPEAT		
			ELSE	// sort ascending
				REPEAT	
					i 										:= i+1;
					pCmpElement								:= pCompareElement + (SizeOfStruct * TO_UDINT(i-1));
				UNTIL (pCmpElement^ >= PivotElement)	OR NOT (i < right)	END_REPEAT;				
				REPEAT	
					j 										:= j-1;	
					pCmpElement								:= pCompareElement + (SizeOfStruct * TO_UDINT(j-1));
				UNTIL (pCmpElement^ <= PivotElement) OR NOT (j > left)	END_REPEAT;
			END_IF
			IF i >= j THEN
				endSubLoop									:= TRUE;
			ELSE                    					
				Allocate(SizeOfStruct);
				pElement_1									:= pData + (SizeOfStruct * TO_UDINT(j-1));
				pElement_2									:= pData + (SizeOfStruct * TO_UDINT(i-1));
				
				IF pElement_Tmp = 0 
					OR_ELSE MEMCPY(pElement_Tmp, pElement_1,	SizeOfStruct) = 0
					OR_ELSE MEMCPY(pElement_1,	pElement_2,		SizeOfStruct) = 0
					OR_ELSE MEMCPY(pElement_2,	pElement_Tmp,	SizeOfStruct) = 0
				THEN
					byUINT									:= FALSE;
					RETURN;	
				END_IF

			END_IF
		UNTIL endSubLoop END_REPEAT;		
		stack[stackCount] 									:= TO_UDINT(right); 	// save right in stack			
		IF stackCount < 32              					
		THEN                            					
			stackCount 										:= stackCount +1;
		ELSE															// Error stack Limit    
			endMainLoop 									:= TRUE;
			byUINT											:= FALSE;			
		END_IF                          					
		right 												:= MAX(left, i-1);
	ELSE                                
		IF stackCount = 1 THEN          
			endMainLoop 									:= TRUE;
		ELSE                            					
			left 											:= right+1;       
			stackCount 										:= stackCount -1;	// load from stack
			right											:= TO_DINT(stack[stackCount]);
		END_IF
	END_IF
END_WHILE
END_METHOD

METHOD byUSINT : BOOL // returns true if sort ends successfully 
VAR_INPUT
	pData													: 	POINTER TO BYTE := 0;	// ADR(Array) 	
	SizeOfData												: 	UDINT := 0;				// SIZEOF(Array)
	pCompareElement											: 	POINTER TO BYTE := 0;	// ADR(Array[1].USINT)		
	SizeOfStruct											: 	UDINT := 0;				// SIZEOF(Array[1]) 	
END_VAR                                                 
VAR        
	pPivotElement											: 	POINTER TO USINT;		// Pivot value	
	PivotElement											: 	USINT;					// Pivot value as USINT
	pCmpElement												:	POINTER TO USINT;		// compare value
	                                					                            	
	endMainLoop												:	BOOL;					// End of main loop reached
	endSubLoop												:	BOOL;					// End of sub loop reached                                              
	ElementCount											:	DINT;					// No of array elements
	stackCount,left,right,i,j								:	DINT;					// running variables 	
	stack													:	ARRAY[1..32] OF UDINT;	// stack size 32 => ~1 Mio elements *)	
	                                					
	pElement_1												:	POINTER TO BYTE;		// Copy Pointer 1		
	pElement_2												:	POINTER TO BYTE;		// Copy Pointer 2
END_VAR
// ends with true in case of no error	                                    					 					
IF SizeOfStruct = 0 OR SizeOfData = 0
	OR pData = 0 OR pCompareElement = 0
THEN               					                                   					
	byUSINT													:= FALSE;
	RETURN;   
ELSE
	byUSINT													:= TRUE;                          					
END_IF    

// calculate no. of Elements                                
ElementCount												:= TO_DINT(SizeOfData / SizeOfStruct);                               					
                                        					
// Quicksort                            					
// initial value of array size          					
left 														:= 1;				// first element
right 														:= ElementCount;	// last element 
stackCount 													:= 1;				// running variable 
                                        	
WHILE NOT endMainLoop DO							
	IF left < right THEN                	
		pPivotElement										:= pCompareElement + (SizeOfStruct * TO_UDINT(SHR(right+left,1)));
		PivotElement										:= pPivotElement^;
		i 													:= left -1;
		j 													:= right +1;
		endSubLoop 											:= FALSE;
		REPEAT
			IF SortInverse
			THEN	// sort descending	
				REPEAT	
					i 										:= i+1;	
					pCmpElement								:= pCompareElement + (SizeOfStruct * TO_UDINT(i-1));
				UNTIL (pCmpElement^ <= PivotElement) OR NOT (i < right)	END_REPEAT	
				REPEAT	
					j 										:= j-1;	
					pCmpElement								:= pCompareElement + (SizeOfStruct * TO_UDINT(j-1));
				UNTIL (pCmpElement^ >= PivotElement) OR NOT (j > left)	END_REPEAT		
			ELSE	// sort ascending
				REPEAT	
					i 										:= i+1;
					pCmpElement								:= pCompareElement + (SizeOfStruct * TO_UDINT(i-1));
				UNTIL (pCmpElement^ >= PivotElement)	OR NOT (i < right)	END_REPEAT;				
				REPEAT	
					j 										:= j-1;	
					pCmpElement								:= pCompareElement + (SizeOfStruct * TO_UDINT(j-1));
				UNTIL (pCmpElement^ <= PivotElement) OR NOT (j > left)	END_REPEAT;
			END_IF
			IF i >= j THEN
				endSubLoop									:= TRUE;
			ELSE                    					
				Allocate(SizeOfStruct);
				pElement_1									:= pData + (SizeOfStruct * TO_UDINT(j-1));
				pElement_2									:= pData + (SizeOfStruct * TO_UDINT(i-1));
				
				IF pElement_Tmp = 0 
					OR_ELSE MEMCPY(pElement_Tmp, pElement_1,	SizeOfStruct) = 0
					OR_ELSE MEMCPY(pElement_1,	pElement_2,		SizeOfStruct) = 0
					OR_ELSE MEMCPY(pElement_2,	pElement_Tmp,	SizeOfStruct) = 0
				THEN
					byUSINT									:= FALSE;
					RETURN;	
				END_IF

			END_IF
		UNTIL endSubLoop END_REPEAT;		
		stack[stackCount] 									:= TO_UDINT(right); 	// save right in stack			
		IF stackCount < 32              					
		THEN                            					
			stackCount 										:= stackCount +1;
		ELSE															// Error stack Limit    
			endMainLoop 									:= TRUE;
			byUSINT											:= FALSE;			
		END_IF                          					
		right 												:= MAX(left, i-1);
	ELSE                                
		IF stackCount = 1 THEN          
			endMainLoop 									:= TRUE;
		ELSE                            					
			left 											:= right+1;       
			stackCount 										:= stackCount -1;	// load from stack
			right											:= TO_DINT(stack[stackCount]);
		END_IF
	END_IF
END_WHILE
END_METHOD

METHOD byWSTRING : BOOL // returns true if sort ends successfully 
VAR_INPUT
	pData													: 	POINTER TO BYTE := 0;	// ADR(Array) 	
	SizeOfData												: 	UDINT := 0;				// SIZEOF(Array)
	pCompareElement											: 	POINTER TO BYTE := 0;	// ADR(Array[1].WSTRING)		
	SizeOfStruct											: 	UDINT := 0;				// SIZEOF(Array[1]) 	
END_VAR                                                                                            
VAR        
	pPivotElement											: 	POINTER TO WSTRING(MAX_WSTRING_LENGTH);	// Pivot value	
	pCmpElement												:	POINTER TO WSTRING(MAX_WSTRING_LENGTH);	// compare value
	PivotElement											:	WORD; 					// Pivot value	
	CompareElement											:	WORD; 					// compare value
	                                					                            	
	endMainLoop												:	BOOL;					// End of main loop reached
	endSubLoop												:	BOOL;					// End of sub loop reached                                              
	ElementCount											:	DINT;					// No of array elements
	stackCount,left,right,i,j,k								:	DINT;					// running variables 	
	stack													:	ARRAY[1..32] OF UDINT;	// stack size 32 => ~1 Mio elements *)	
	                                					
	pElement_1												:	POINTER TO BYTE;		// Copy Pointer 1		
	pElement_2												:	POINTER TO BYTE;		// Copy Pointer 2
END_VAR
// ends with true in case of no error	                                    					 					
IF SizeOfStruct = 0 OR SizeOfData = 0
	OR pData = 0 OR pCompareElement = 0
THEN               					                                   					
	byWSTRING												:= FALSE;
	RETURN;   
ELSE
	byWSTRING												:= TRUE;                          					
END_IF                                   					
            
// calculate no. of Elements                                
ElementCount												:= TO_DINT(SizeOfData / SizeOfStruct);   
                            					
// Quicksort                            					
// initial value of array size          					
left 														:= 1;				// first element
right 														:= ElementCount;	// last element 
stackCount 													:= 1;				// running variable 
                                        	
